# B&R Automation Studio project Kontrol (part 2)

#### Cyclic.st
```iecst
PROGRAM _CYCLIC

	//-------------------------------------------------------------------------------------------
	(*Parametros*)
	IF link_mdb_parametros.NewValue THEN
		link_mdb_parametros.NewValue    := FALSE;
	//-------------------------------------------------------------------------------------------

		UG.Parametro.UP_Partindo_Tempo := MDB_Parametros[1];
		UG.Parametro.UPGM_Partindo_Tempo := MDB_Parametros[2];
		UG.Parametro.UMVD_Partindo_Tempo := MDB_Parametros[3];
		UG.Parametro.UPS_Partindo_Tempo := MDB_Parametros[4];
		UG.Parametro.US_Parando_Tempo := MDB_Parametros[5];
		UG.Parametro.UPS_Parando_Tempo := MDB_Parametros[6];
		UG.Parametro.UMVD_Parando_Tempo := MDB_Parametros[7];
		UG.Parametro.UPGM_Parando_Tempo := MDB_Parametros[8];
		UG.Parametro.UPGM_Fechar_FA_Tempo := MDB_Parametros[9];
		//0.0 := MDB_Parametros[10];
		//0.0 := MDB_Parametros[11];
		//0.0 := MDB_Parametros[12];
		//0.0 := MDB_Parametros[13];
		//0.0 := MDB_Parametros[14];
		//0.0 := MDB_Parametros[15];
		//0.0 := MDB_Parametros[16];
		//0.0 := MDB_Parametros[17];
		//0.0 := MDB_Parametros[18];
		//0.0 := MDB_Parametros[19];
		//0.0 := MDB_Parametros[20];
		SFA.Parametro.Delta_Pressao.SensorMin := MDB_Parametros[21];
		SFA.Parametro.Delta_Pressao.SensorMax := MDB_Parametros[22];
		SFA.Parametro.Delta_Pressao.Alarme := MDB_Parametros[23];
		SFA.Parametro.Delta_Pressao.Trip := MDB_Parametros[24];
		SFA.Parametro.Delta_Pressao.Tempo_AL := MDB_Parametros[25];
		SFA.Parametro.Delta_Pressao.Tempo_TR := MDB_Parametros[26];
		SFA.Parametro.Pressao1_Lado_Limpo.SensorMin := MDB_Parametros[27];
		SFA.Parametro.Pressao1_Lado_Limpo.SensorMax := MDB_Parametros[28];
		SFA.Parametro.Pressao1_Lado_Limpo.Alarme := MDB_Parametros[29];
		SFA.Parametro.Pressao1_Lado_Limpo.Trip := MDB_Parametros[30];
		SFA.Parametro.Pressao1_Lado_Limpo.Tempo_AL := MDB_Parametros[31];
		SFA.Parametro.Pressao1_Lado_Limpo.Tempo_TR := MDB_Parametros[32];
		SFA.Parametro.Pressao2_Lado_Limpo.SensorMin := MDB_Parametros[33];
		SFA.Parametro.Pressao2_Lado_Limpo.SensorMax := MDB_Parametros[34];
		SFA.Parametro.Pressao2_Lado_Limpo.Alarme := MDB_Parametros[35];
		SFA.Parametro.Pressao2_Lado_Limpo.Trip := MDB_Parametros[36];
		SFA.Parametro.Pressao2_Lado_Limpo.Tempo_AL := MDB_Parametros[37];
		SFA.Parametro.Pressao2_Lado_Limpo.Tempo_TR := MDB_Parametros[38];
		SFA.Parametro.Pressao1_Lado_Sujo.SensorMin := MDB_Parametros[39];
		SFA.Parametro.Pressao1_Lado_Sujo.SensorMax := MDB_Parametros[40];
		SFA.Parametro.Pressao1_Lado_Sujo.Alarme := MDB_Parametros[41];
		SFA.Parametro.Pressao1_Lado_Sujo.Trip := MDB_Parametros[42];
		SFA.Parametro.Pressao1_Lado_Sujo.Tempo_AL := MDB_Parametros[43];
		SFA.Parametro.Pressao1_Lado_Sujo.Tempo_TR := MDB_Parametros[44];
		SFA.Parametro.Pressao2_Lado_Sujo.SensorMin := MDB_Parametros[45];
		SFA.Parametro.Pressao2_Lado_Sujo.SensorMax := MDB_Parametros[46];
		SFA.Parametro.Pressao2_Lado_Sujo.Alarme := MDB_Parametros[47];
		SFA.Parametro.Pressao2_Lado_Sujo.Trip := MDB_Parametros[48];
		SFA.Parametro.Pressao2_Lado_Sujo.Tempo_AL := MDB_Parametros[49];
		SFA.Parametro.Pressao2_Lado_Sujo.Tempo_TR := MDB_Parametros[50];
		SFA.Parametro.Filtro1_Tempo_Trabalho := MDB_Parametros[51];
		SFA.Parametro.Filtro1_Tempo_Lavagem := MDB_Parametros[52];
		SFA.Parametro.Filtro1_Tempo_Abrir_Filtro_Limpo := MDB_Parametros[53];
		SFA.Parametro.Filtro1_Tempo_Fechar_Filtro_Sujo := MDB_Parametros[54];
		SFA.Parametro.Filtro2_Tempo_Trabalho := MDB_Parametros[55];
		SFA.Parametro.Filtro2_Tempo_Lavagem := MDB_Parametros[56];
		SFA.Parametro.Filtro2_Tempo_Abrir_Filtro_Limpo := MDB_Parametros[57];
		SFA.Parametro.Filtro2_Tempo_Fechar_Filtro_Sujo := MDB_Parametros[58];
		SFA.Parametro.Filtro1_Delta_Retrolav := MDB_Parametros[59]; //delta de pressão para retrolavagem filtro 1
		SFA.Parametro.Filtro2_Delta_Retrolav := MDB_Parametros[60]; //delta de pressão para retrolavagem filtro 2
		//0.0 := MDB_Parametros[61];
		//0.0 := MDB_Parametros[62];
		//0.0 := MDB_Parametros[63];
		//0.0 := MDB_Parametros[64];
		//0.0 := MDB_Parametros[65];
		//0.0 := MDB_Parametros[66];
		//0.0 := MDB_Parametros[67];
		//0.0 := MDB_Parametros[68];
		//0.0 := MDB_Parametros[69];
		//0.0 := MDB_Parametros[70];
		UHLM.Parametro.Temperatura.SensorMin := MDB_Parametros[71];
		UHLM.Parametro.Temperatura.SensorMax := MDB_Parametros[72];
		UHLM.Parametro.Temperatura.Alarme := MDB_Parametros[73];
		UHLM.Parametro.Temperatura.Trip := MDB_Parametros[74];
		UHLM.Parametro.Temperatura.Tempo_AL := MDB_Parametros[75];
		UHLM.Parametro.Temperatura.Tempo_TR := MDB_Parametros[76];
		UHLM.Parametro.Vazao.SensorMin := MDB_Parametros[77];
		UHLM.Parametro.Vazao.SensorMax := MDB_Parametros[78];
		UHLM.Parametro.Vazao.Alarme := MDB_Parametros[79];
		UHLM.Parametro.Vazao.Trip := MDB_Parametros[80];
		UHLM.Parametro.Vazao.Tempo_AL := MDB_Parametros[81];
		UHLM.Parametro.Vazao.Tempo_TR := MDB_Parametros[82];
		UHLM.Parametro.Ventilador.Ligar := MDB_Parametros[83];
		UHLM.Parametro.Ventilador.Desligar := MDB_Parametros[84];
		//0.0 := MDB_Parametros[85];
		//0.0 := MDB_Parametros[86];
		//0.0 := MDB_Parametros[87];
		//0.0 := MDB_Parametros[88];
		//0.0 := MDB_Parametros[89];
		//0.0 := MDB_Parametros[90];
		//0.0 := MDB_Parametros[91];
		//0.0 := MDB_Parametros[92];
		//0.0 := MDB_Parametros[93];
		//0.0 := MDB_Parametros[94];
		//0.0 := MDB_Parametros[95];
		//0.0 := MDB_Parametros[96];
		//0.0 := MDB_Parametros[97];
		//0.0 := MDB_Parametros[98];
		//0.0 := MDB_Parametros[99];
		//0.0 := MDB_Parametros[100];
		UHRV.Parametro.Temperatura.SensorMin := MDB_Parametros[101];
		UHRV.Parametro.Temperatura.SensorMax := MDB_Parametros[102];
		UHRV.Parametro.Temperatura.Alarme := MDB_Parametros[103];
		UHRV.Parametro.Temperatura.Trip := MDB_Parametros[104];
		UHRV.Parametro.Temperatura.Tempo_AL := MDB_Parametros[105];
		UHRV.Parametro.Temperatura.Tempo_TR := MDB_Parametros[106];
		UHRV.Parametro.Pressao.SensorMin := MDB_Parametros[107];
		UHRV.Parametro.Pressao.SensorMax := MDB_Parametros[108];
		UHRV.Parametro.Pressao.Alarme := MDB_Parametros[109];
		UHRV.Parametro.Pressao.Trip := MDB_Parametros[110];
		UHRV.Parametro.Pressao.Tempo_AL := MDB_Parametros[111];
		UHRV.Parametro.Pressao.Tempo_TR := MDB_Parametros[112];
		UHRV.Parametro.Pressao.Normal_Min := MDB_Parametros[113];
		UHRV.Parametro.Pressao.Normal_Max := MDB_Parametros[114];
		UHRV.Parametro.Tempo_Pressurizar := MDB_Parametros[115];
		//0.0 := MDB_Parametros[116];
		//0.0 := MDB_Parametros[117];
		//0.0 := MDB_Parametros[118];
		//0.0 := MDB_Parametros[119];
		//0.0 := MDB_Parametros[120];
		//0.0 := MDB_Parametros[121];
		//0.0 := MDB_Parametros[122];
		//0.0 := MDB_Parametros[123];
		//0.0 := MDB_Parametros[124];
		//0.0 := MDB_Parametros[125];
		//0.0 := MDB_Parametros[126];
		//0.0 := MDB_Parametros[127];
		//0.0 := MDB_Parametros[128];
		//0.0 := MDB_Parametros[129];
		//0.0 := MDB_Parametros[130];
		Freio.Parametro.Tempo_Aplicado := MDB_Parametros[131];
		Freio.Parametro.Tempo_Desaplicado := MDB_Parametros[132];
		//0.0 := MDB_Parametros[133];
		//0.0 := MDB_Parametros[134];
		//0.0 := MDB_Parametros[135];
		//0.0 := MDB_Parametros[136];
		//0.0 := MDB_Parametros[137];
		//0.0 := MDB_Parametros[138];
		//0.0 := MDB_Parametros[139];
		//0.0 := MDB_Parametros[140];
//		VByPass.Parametro.Tempo.Abrir := MDB_Parametros[141];
//		VByPass.Parametro.Tempo.Fechar := MDB_Parametros[142];
		//0.0 := MDB_Parametros[143];
		//0.0 := MDB_Parametros[144];
		//0.0 := MDB_Parametros[145];
		//0.0 := MDB_Parametros[146];
		//0.0 := MDB_Parametros[147];
		//0.0 := MDB_Parametros[148];
		//0.0 := MDB_Parametros[149];
		//0.0 := MDB_Parametros[150];
//		VBorb.Parametro.Tempo.Abrir := MDB_Parametros[151];
//		VBorb.Parametro.Tempo.Fechar := MDB_Parametros[152];
//		VBorb.Parametro.Tempo.Equalizar := MDB_Parametros[153];
//		VBorb.Parametro.Delta_Pressao := MDB_Parametros[154];
//		VBorb.Parametro.Pressao.Montante.SensorMin := MDB_Parametros[155];
//		VBorb.Parametro.Pressao.Montante.SensorMax := MDB_Parametros[156];
//		VBorb.Parametro.Pressao.Jusante.SensorMin := MDB_Parametros[157];
//		VBorb.Parametro.Pressao.Jusante.SensorMax := MDB_Parametros[158];
		//0.0 := MDB_Parametros[159];
		//0.0 := MDB_Parametros[160];
		//0.0 := MDB_Parametros[161];
		//0.0 := MDB_Parametros[162];
		//0.0 := MDB_Parametros[163];
		//0.0 := MDB_Parametros[164];
		//0.0 := MDB_Parametros[165];
		//0.0 := MDB_Parametros[166];
		//0.0 := MDB_Parametros[167];
		Comporta1.Parametro.Encoder1_SensorMin := MDB_Parametros[168];
		Comporta1.Parametro.Encoder1_SensorMax := MDB_Parametros[169];
		Comporta1.Parametro.Tempo_Cracking := MDB_Parametros[170];
		Comporta1.Parametro.Tempo_Falha_Abertura := MDB_Parametros[171];
		Comporta1.Parametro.Tempo_Falha_Cracking := MDB_Parametros[172];
		Comporta1.Parametro.Tempo_Falha_Fechando := MDB_Parametros[173];
		Comporta1.Parametro.Tempo_Falha_Reposicao := MDB_Parametros[174];
//		Comporta.Parametro.Pressao.Montante.SensorMin := MDB_Parametros[175];
//		Comporta.Parametro.Pressao.Montante.SensorMax := MDB_Parametros[176];
		Comporta2.Parametro.Encoder2_SensorMin := MDB_Parametros[177];
		Comporta2.Parametro.Encoder2_SensorMax := MDB_Parametros[178];
		Comporta2.Parametro.Tempo_Cracking := MDB_Parametros[179];
		Comporta2.Parametro.Tempo_Falha_Abertura := MDB_Parametros[180];
		Comporta2.Parametro.Tempo_Falha_Cracking := MDB_Parametros[181];
		Comporta2.Parametro.Tempo_Falha_Fechando := MDB_Parametros[182];
		Comporta2.Parametro.Tempo_Falha_Reposicao := MDB_Parametros[183];
		Comporta_UH.Parametro.Temperatura_Oleo.SensorMin := MDB_Parametros[184];
		Comporta_UH.Parametro.Temperatura_Oleo.SensorMax := MDB_Parametros[185];
		Comporta_UH.Parametro.Temperatura_Oleo.Alarme := MDB_Parametros[186];
		Comporta_UH.Parametro.Temperatura_Oleo.Trip := MDB_Parametros[187];
		Comporta_UH.Parametro.Temperatura_Oleo.Tempo_AL := MDB_Parametros[188];
		Comporta_UH.Parametro.Temperatura_Oleo.Tempo_TR := MDB_Parametros[189];
		//0.0 := MDB_Parametros[190];
		Turbina.Parametro.Gaxeteiro.Temperatura.SensorMin := MDB_Parametros[191];
		Turbina.Parametro.Gaxeteiro.Temperatura.SensorMax := MDB_Parametros[192];
		Turbina.Parametro.Gaxeteiro.Temperatura.Alarme := MDB_Parametros[193];
		Turbina.Parametro.Gaxeteiro.Temperatura.Trip := MDB_Parametros[194];
		Turbina.Parametro.Gaxeteiro.Temperatura.Tempo_AL := MDB_Parametros[195];
		Turbina.Parametro.Gaxeteiro.Temperatura.Tempo_TR := MDB_Parametros[196];
		Turbina.Parametro.Mancal1.Temperatura.SensorMin := MDB_Parametros[197];
		Turbina.Parametro.Mancal1.Temperatura.SensorMax := MDB_Parametros[198];
		Turbina.Parametro.Mancal1.Temperatura.Alarme := MDB_Parametros[199];
		Turbina.Parametro.Mancal1.Temperatura.Trip := MDB_Parametros[200];
		Turbina.Parametro.Mancal1.Temperatura.Tempo_AL := MDB_Parametros[201];
		Turbina.Parametro.Mancal1.Temperatura.Tempo_TR := MDB_Parametros[202];
		Turbina.Parametro.Mancal2.Temperatura.SensorMin := MDB_Parametros[203];
		Turbina.Parametro.Mancal2.Temperatura.SensorMax := MDB_Parametros[204];
		Turbina.Parametro.Mancal2.Temperatura.Alarme := MDB_Parametros[205];
		Turbina.Parametro.Mancal2.Temperatura.Trip := MDB_Parametros[206];
		Turbina.Parametro.Mancal2.Temperatura.Tempo_AL := MDB_Parametros[207];
		Turbina.Parametro.Mancal2.Temperatura.Tempo_TR := MDB_Parametros[208];
		Turbina.Parametro.Mancal3.Temperatura.SensorMin := MDB_Parametros[209];
		Turbina.Parametro.Mancal3.Temperatura.SensorMax := MDB_Parametros[210];
		Turbina.Parametro.Mancal3.Temperatura.Alarme := MDB_Parametros[211];
		Turbina.Parametro.Mancal3.Temperatura.Trip := MDB_Parametros[212];
		Turbina.Parametro.Mancal3.Temperatura.Tempo_AL := MDB_Parametros[213];
		Turbina.Parametro.Mancal3.Temperatura.Tempo_TR := MDB_Parametros[214];
		Turbina.Parametro.Mancal4.Temperatura.SensorMin := MDB_Parametros[215];
		Turbina.Parametro.Mancal4.Temperatura.SensorMax := MDB_Parametros[216];
		Turbina.Parametro.Mancal4.Temperatura.Alarme := MDB_Parametros[217];
		Turbina.Parametro.Mancal4.Temperatura.Trip := MDB_Parametros[218];
		Turbina.Parametro.Mancal4.Temperatura.Tempo_AL := MDB_Parametros[219];
		Turbina.Parametro.Mancal4.Temperatura.Tempo_TR := MDB_Parametros[220];
		Turbina.Parametro.Mancal5.Temperatura.SensorMin := MDB_Parametros[221];
		Turbina.Parametro.Mancal5.Temperatura.SensorMax := MDB_Parametros[222];
		Turbina.Parametro.Mancal5.Temperatura.Alarme := MDB_Parametros[223];
		Turbina.Parametro.Mancal5.Temperatura.Trip := MDB_Parametros[224];
		Turbina.Parametro.Mancal5.Temperatura.Tempo_AL := MDB_Parametros[225];
		Turbina.Parametro.Mancal5.Temperatura.Tempo_TR := MDB_Parametros[226];
		Turbina.Parametro.Mancal6.Temperatura.SensorMin := MDB_Parametros[227];
		Turbina.Parametro.Mancal6.Temperatura.SensorMax := MDB_Parametros[228];
		Turbina.Parametro.Mancal6.Temperatura.Alarme := MDB_Parametros[229];
		Turbina.Parametro.Mancal6.Temperatura.Trip := MDB_Parametros[230];
		Turbina.Parametro.Mancal6.Temperatura.Tempo_AL := MDB_Parametros[231];
		Turbina.Parametro.Mancal6.Temperatura.Tempo_TR := MDB_Parametros[232];
		Turbina.Parametro.CaixaEspiral.Pressao.SensorMin := MDB_Parametros[233];
		Turbina.Parametro.CaixaEspiral.Pressao.SensorMax := MDB_Parametros[234];
		Turbina.Parametro.CaixaEspiral.Pressao.Alarme := MDB_Parametros[235];
		Turbina.Parametro.CaixaEspiral.Pressao.Trip := MDB_Parametros[236];
		Turbina.Parametro.CaixaEspiral.Pressao.Tempo_AL := MDB_Parametros[237];
		Turbina.Parametro.CaixaEspiral.Pressao.Tempo_TR := MDB_Parametros[238];
		Turbina.Parametro.Delta_Pressao := MDB_Parametros[239];
		//0.0 := MDB_Parametros[240];
		//0.0 := MDB_Parametros[241];
		//0.0 := MDB_Parametros[242];
		//0.0 := MDB_Parametros[243];
		//0.0 := MDB_Parametros[244];
		//0.0 := MDB_Parametros[245];
		//0.0 := MDB_Parametros[246];
		//0.0 := MDB_Parametros[247];
		//0.0 := MDB_Parametros[248];
		//0.0 := MDB_Parametros[249];
		//0.0 := MDB_Parametros[250];
		Gerador.Parametro.Fase_A.Temperatura.SensorMin := MDB_Parametros[251];
		Gerador.Parametro.Fase_A.Temperatura.SensorMax := MDB_Parametros[252];
		Gerador.Parametro.Fase_A.Temperatura.Alarme := MDB_Parametros[253];
		Gerador.Parametro.Fase_A.Temperatura.Trip := MDB_Parametros[254];
		Gerador.Parametro.Fase_A.Temperatura.Tempo_AL := MDB_Parametros[255];
		Gerador.Parametro.Fase_A.Temperatura.Tempo_TR := MDB_Parametros[256];
		Gerador.Parametro.Fase_B.Temperatura.SensorMin := MDB_Parametros[257];
		Gerador.Parametro.Fase_B.Temperatura.SensorMax := MDB_Parametros[258];
		Gerador.Parametro.Fase_B.Temperatura.Alarme := MDB_Parametros[259];
		Gerador.Parametro.Fase_B.Temperatura.Trip := MDB_Parametros[260];
		Gerador.Parametro.Fase_B.Temperatura.Tempo_AL := MDB_Parametros[261];
		Gerador.Parametro.Fase_B.Temperatura.Tempo_TR := MDB_Parametros[262];
		Gerador.Parametro.Fase_C.Temperatura.SensorMin := MDB_Parametros[263];
		Gerador.Parametro.Fase_C.Temperatura.SensorMax := MDB_Parametros[264];
		Gerador.Parametro.Fase_C.Temperatura.Alarme := MDB_Parametros[265];
		Gerador.Parametro.Fase_C.Temperatura.Trip := MDB_Parametros[266];
		Gerador.Parametro.Fase_C.Temperatura.Tempo_AL := MDB_Parametros[267];
		Gerador.Parametro.Fase_C.Temperatura.Tempo_TR := MDB_Parametros[268];
		Gerador.Parametro.NucleoEstatorico1.Temperatura.SensorMin := MDB_Parametros[269];
		Gerador.Parametro.NucleoEstatorico1.Temperatura.SensorMax := MDB_Parametros[270];
		Gerador.Parametro.NucleoEstatorico1.Temperatura.Alarme := MDB_Parametros[271];
		Gerador.Parametro.NucleoEstatorico1.Temperatura.Trip := MDB_Parametros[272];
		Gerador.Parametro.NucleoEstatorico1.Temperatura.Tempo_AL := MDB_Parametros[273];
		Gerador.Parametro.NucleoEstatorico1.Temperatura.Tempo_TR := MDB_Parametros[274];
		Gerador.Parametro.NucleoEstatorico2.Temperatura.SensorMin := MDB_Parametros[275];
		Gerador.Parametro.NucleoEstatorico2.Temperatura.SensorMax := MDB_Parametros[276];
		Gerador.Parametro.NucleoEstatorico2.Temperatura.Alarme := MDB_Parametros[277];
		Gerador.Parametro.NucleoEstatorico2.Temperatura.Trip := MDB_Parametros[278];
		Gerador.Parametro.NucleoEstatorico2.Temperatura.Tempo_AL := MDB_Parametros[279];
		Gerador.Parametro.NucleoEstatorico2.Temperatura.Tempo_TR := MDB_Parametros[280];
		Gerador.Parametro.NucleoEstatorico3.Temperatura.SensorMin := MDB_Parametros[281];
		Gerador.Parametro.NucleoEstatorico3.Temperatura.SensorMax := MDB_Parametros[282];
		Gerador.Parametro.NucleoEstatorico3.Temperatura.Alarme := MDB_Parametros[283];
		Gerador.Parametro.NucleoEstatorico3.Temperatura.Trip := MDB_Parametros[284];
		Gerador.Parametro.NucleoEstatorico3.Temperatura.Tempo_AL := MDB_Parametros[285];
		Gerador.Parametro.NucleoEstatorico3.Temperatura.Tempo_TR := MDB_Parametros[286];
		Gerador.Parametro.Mancal1.Temperatura.SensorMin := MDB_Parametros[287];
		Gerador.Parametro.Mancal1.Temperatura.SensorMax := MDB_Parametros[288];
		Gerador.Parametro.Mancal1.Temperatura.Alarme := MDB_Parametros[289];
		Gerador.Parametro.Mancal1.Temperatura.Trip := MDB_Parametros[290];
		Gerador.Parametro.Mancal1.Temperatura.Tempo_AL := MDB_Parametros[291];
		Gerador.Parametro.Mancal1.Temperatura.Tempo_TR := MDB_Parametros[292];
		Gerador.Parametro.Mancal2.Temperatura.SensorMin := MDB_Parametros[293];
		Gerador.Parametro.Mancal2.Temperatura.SensorMax := MDB_Parametros[294];
		Gerador.Parametro.Mancal2.Temperatura.Alarme := MDB_Parametros[295];
		Gerador.Parametro.Mancal2.Temperatura.Trip := MDB_Parametros[296];
		Gerador.Parametro.Mancal2.Temperatura.Tempo_AL := MDB_Parametros[297];
		Gerador.Parametro.Mancal2.Temperatura.Tempo_TR := MDB_Parametros[298];
		Gerador.Parametro.Mancal3.Temperatura.SensorMin := MDB_Parametros[299];
		Gerador.Parametro.Mancal3.Temperatura.SensorMax := MDB_Parametros[300];
		Gerador.Parametro.Mancal3.Temperatura.Alarme := MDB_Parametros[301];
		Gerador.Parametro.Mancal3.Temperatura.Trip := MDB_Parametros[302];
		Gerador.Parametro.Mancal3.Temperatura.Tempo_AL := MDB_Parametros[303];
		Gerador.Parametro.Mancal3.Temperatura.Tempo_TR := MDB_Parametros[304];
		Gerador.Parametro.Mancal4.Temperatura.SensorMin := MDB_Parametros[305];
		Gerador.Parametro.Mancal4.Temperatura.SensorMax := MDB_Parametros[306];
		Gerador.Parametro.Mancal4.Temperatura.Alarme := MDB_Parametros[307];
		Gerador.Parametro.Mancal4.Temperatura.Trip := MDB_Parametros[308];
		Gerador.Parametro.Mancal4.Temperatura.Tempo_AL := MDB_Parametros[309];
		Gerador.Parametro.Mancal4.Temperatura.Tempo_TR := MDB_Parametros[310];
		Gerador.Parametro.Mancal5.Temperatura.SensorMin := MDB_Parametros[311];
		Gerador.Parametro.Mancal5.Temperatura.SensorMax := MDB_Parametros[312];
		Gerador.Parametro.Mancal5.Temperatura.Alarme := MDB_Parametros[313];
		Gerador.Parametro.Mancal5.Temperatura.Trip := MDB_Parametros[314];
		Gerador.Parametro.Mancal5.Temperatura.Tempo_AL := MDB_Parametros[315];
		Gerador.Parametro.Mancal5.Temperatura.Tempo_TR := MDB_Parametros[316];
		Gerador.Parametro.Mancal6.Temperatura.SensorMin := MDB_Parametros[317];
		Gerador.Parametro.Mancal6.Temperatura.SensorMax := MDB_Parametros[318];
		Gerador.Parametro.Mancal6.Temperatura.Alarme := MDB_Parametros[319];
		Gerador.Parametro.Mancal6.Temperatura.Trip := MDB_Parametros[320];
		Gerador.Parametro.Mancal6.Temperatura.Tempo_AL := MDB_Parametros[321];
		Gerador.Parametro.Mancal6.Temperatura.Tempo_TR := MDB_Parametros[322];
		//0.0 := MDB_Parametros[323];
		//0.0 := MDB_Parametros[324];
		//0.0 := MDB_Parametros[325];
		//0.0 := MDB_Parametros[326];
		//0.0 := MDB_Parametros[327];
		//0.0 := MDB_Parametros[328];
		//0.0 := MDB_Parametros[329];
		//0.0 := MDB_Parametros[330];
		//0.0 := MDB_Parametros[331];
		//0.0 := MDB_Parametros[332];
		//0.0 := MDB_Parametros[333];
		//0.0 := MDB_Parametros[334];
		//0.0 := MDB_Parametros[335];
		//0.0 := MDB_Parametros[336];
		//0.0 := MDB_Parametros[337];
		//0.0 := MDB_Parametros[338];
		//0.0 := MDB_Parametros[339];
		//0.0 := MDB_Parametros[340];
		RT.Parametro.PWR.Temperatura.SensorMin := MDB_Parametros[341];
		RT.Parametro.PWR.Temperatura.SensorMax := MDB_Parametros[342];
		RT.Parametro.PWR.Temperatura.Alarme := MDB_Parametros[343];
		RT.Parametro.PWR.Temperatura.Trip := MDB_Parametros[344];
		RT.Parametro.PWR.Temperatura.Tempo_AL := MDB_Parametros[345];
		RT.Parametro.PWR.Temperatura.Tempo_TR := MDB_Parametros[346];
		//0.0 := MDB_Parametros[347];
		//0.0 := MDB_Parametros[348];
		//0.0 := MDB_Parametros[349];
		//0.0 := MDB_Parametros[350];
		//0.0 := MDB_Parametros[351];
		//0.0 := MDB_Parametros[352];
		//0.0 := MDB_Parametros[353];
		//0.0 := MDB_Parametros[354];
		//0.0 := MDB_Parametros[355];
		//0.0 := MDB_Parametros[356];
		//0.0 := MDB_Parametros[357];
		//0.0 := MDB_Parametros[358];
		//0.0 := MDB_Parametros[359];
		//0.0 := MDB_Parametros[360];
		Trafo_Exc.Parametro.Fase_A.Temperatura.SensorMin := MDB_Parametros[361];
		Trafo_Exc.Parametro.Fase_A.Temperatura.SensorMax := MDB_Parametros[362];
		Trafo_Exc.Parametro.Fase_A.Temperatura.Alarme := MDB_Parametros[363];
		Trafo_Exc.Parametro.Fase_A.Temperatura.Trip := MDB_Parametros[364];
		Trafo_Exc.Parametro.Fase_A.Temperatura.Tempo_AL := MDB_Parametros[365];
		Trafo_Exc.Parametro.Fase_A.Temperatura.Tempo_TR := MDB_Parametros[366];
		Trafo_Exc.Parametro.Fase_B.Temperatura.SensorMin := MDB_Parametros[367];
		Trafo_Exc.Parametro.Fase_B.Temperatura.SensorMax := MDB_Parametros[368];
		Trafo_Exc.Parametro.Fase_B.Temperatura.Alarme := MDB_Parametros[369];
		Trafo_Exc.Parametro.Fase_B.Temperatura.Trip := MDB_Parametros[370];
		Trafo_Exc.Parametro.Fase_B.Temperatura.Tempo_AL := MDB_Parametros[371];
		Trafo_Exc.Parametro.Fase_B.Temperatura.Tempo_TR := MDB_Parametros[372];
		Trafo_Exc.Parametro.Fase_C.Temperatura.SensorMin := MDB_Parametros[373];
		Trafo_Exc.Parametro.Fase_C.Temperatura.SensorMax := MDB_Parametros[374];
		Trafo_Exc.Parametro.Fase_C.Temperatura.Alarme := MDB_Parametros[375];
		Trafo_Exc.Parametro.Fase_C.Temperatura.Trip := MDB_Parametros[376];
		Trafo_Exc.Parametro.Fase_C.Temperatura.Tempo_AL := MDB_Parametros[377];
		Trafo_Exc.Parametro.Fase_C.Temperatura.Tempo_TR := MDB_Parametros[378];
		//0.0 := MDB_Parametros[379];
		//0.0 := MDB_Parametros[380];
		//0.0 := MDB_Parametros[381];
		//0.0 := MDB_Parametros[382];
		//0.0 := MDB_Parametros[383];
		//0.0 := MDB_Parametros[384];
		//0.0 := MDB_Parametros[385];
		//0.0 := MDB_Parametros[386];
		//0.0 := MDB_Parametros[387];
		//0.0 := MDB_Parametros[388];
		//0.0 := MDB_Parametros[389];
		//0.0 := MDB_Parametros[390];
		Nivel.Parametro.Nivel_Ligar := MDB_Parametros[391];
		Nivel.Parametro.Nivel_Desligar := MDB_Parametros[392];
		Nivel.Parametro.Nivel_Trip := MDB_Parametros[393];
		Nivel.Parametro.Nivel_Min := MDB_Parametros[394];
		Nivel.Parametro.Nivel_Max := MDB_Parametros[395];
		Nivel.Parametro.Potencia_Min := MDB_Parametros[396];
		Nivel.Parametro.Potencia_Max := MDB_Parametros[397];
		Nivel.Parametro.PID.Kp := MDB_Parametros[398];
		Nivel.Parametro.PID.Ki := MDB_Parametros[399];
		Nivel.Parametro.PID.Kd := MDB_Parametros[400];
		Nivel.Parametro.PID.Tf := MDB_Parametros[401];
		//0.0 := MDB_Parametros[402];
		//0.0 := MDB_Parametros[403];
		//0.0 := MDB_Parametros[404];
		//0.0 := MDB_Parametros[405];
		//0.0 := MDB_Parametros[406];
		//0.0 := MDB_Parametros[407];
		//0.0 := MDB_Parametros[408];
		//0.0 := MDB_Parametros[409];
		//0.0 := MDB_Parametros[410];
		Nivel.Parametro.Barragem.SensorMin := MDB_Parametros[411];
		Nivel.Parametro.Barragem.SensorMax := MDB_Parametros[412];
		//0.0 := MDB_Parametros[413];
		//0.0 := MDB_Parametros[414];
		Nivel.Parametro.Barragem.Alarme := MDB_Parametros[415];
		Nivel.Parametro.Barragem.Trip := MDB_Parametros[416];
		Nivel.Parametro.Barragem.Tempo_AL := MDB_Parametros[417];
		Nivel.Parametro.Barragem.Tempo_TR := MDB_Parametros[418];
		Nivel.Parametro.Jusante.SensorMin := MDB_Parametros[419];
		Nivel.Parametro.Jusante.SensorMax := MDB_Parametros[420];
		//0.0 := MDB_Parametros[421];
		Nivel.Parametro.Jusante.Cota := MDB_Parametros[422];
		Nivel.Parametro.Jusante.Alarme := MDB_Parametros[423];
		Nivel.Parametro.Jusante.Trip := MDB_Parametros[424];
		Nivel.Parametro.Jusante.Tempo_AL := MDB_Parametros[425];
		Nivel.Parametro.Jusante.Tempo_TR := MDB_Parametros[426];
		//0.0 := MDB_Parametros[427];
		//0.0 := MDB_Parametros[428];
		//0.0 := MDB_Parametros[429];
		Nivel.Parametro.Jusante_Grade1.SensorMin := MDB_Parametros[430];
		Nivel.Parametro.Jusante_Grade1.SensorMax := MDB_Parametros[431];
		Nivel.Parametro.Jusante_Grade1.Cota := MDB_Parametros[432];
		Nivel.Parametro.Jusante_Grade1.Alarme := MDB_Parametros[433];
		Nivel.Parametro.Jusante_Grade1.Trip := MDB_Parametros[434];
		Nivel.Parametro.Jusante_Grade1.Tempo_AL := MDB_Parametros[435];
		Nivel.Parametro.Jusante_Grade1.Tempo_TR := MDB_Parametros[436];
		//0.0 := MDB_Parametros[437];
		//0.0 := MDB_Parametros[438];
		//0.0 := MDB_Parametros[439];
		Nivel.Parametro.Jusante_Grade2.SensorMin := MDB_Parametros[440];
		Nivel.Parametro.Jusante_Grade2.SensorMax := MDB_Parametros[441];
		Nivel.Parametro.Jusante_Grade2.Cota := MDB_Parametros[442];
		Nivel.Parametro.Jusante_Grade2.Alarme := MDB_Parametros[443];
		Nivel.Parametro.Jusante_Grade2.Trip := MDB_Parametros[444];
		Nivel.Parametro.Jusante_Grade2.Tempo_AL := MDB_Parametros[445];
		Nivel.Parametro.Jusante_Grade2.Tempo_TR := MDB_Parametros[446];
		//0.0 := MDB_Parametros[447];
		//0.0 := MDB_Parametros[448];
		//0.0 := MDB_Parametros[449];
		//0.0 := MDB_Parametros[450];
		//0.0 := MDB_Parametros[451];
		//0.0 := MDB_Parametros[452];
		//0.0 := MDB_Parametros[453];
		//0.0 := MDB_Parametros[454];
		//0.0 := MDB_Parametros[455];
		//0.0 := MDB_Parametros[456];
		//0.0 := MDB_Parametros[457];
		//0.0 := MDB_Parametros[458];
		//0.0 := MDB_Parametros[459];
		//0.0 := MDB_Parametros[460];

	//-------------------------------------------------------------------------------------------

	ELSE

	//-------------------------------------------------------------------------------------------

		MDB_Parametros[1]:=UG.Parametro.UP_Partindo_Tempo;
		MDB_Parametros[2]:=UG.Parametro.UPGM_Partindo_Tempo;
		MDB_Parametros[3]:=UG.Parametro.UMVD_Partindo_Tempo;
		MDB_Parametros[4]:=UG.Parametro.UPS_Partindo_Tempo;
		MDB_Parametros[5]:=UG.Parametro.US_Parando_Tempo;
		MDB_Parametros[6]:=UG.Parametro.UPS_Parando_Tempo;
		MDB_Parametros[7]:=UG.Parametro.UMVD_Parando_Tempo;
		MDB_Parametros[8]:=UG.Parametro.UPGM_Parando_Tempo;
		MDB_Parametros[9]:=UG.Parametro.UPGM_Fechar_FA_Tempo;
		MDB_Parametros[10]:=0.0;
		MDB_Parametros[11]:=0.0;
		MDB_Parametros[12]:=0.0;
		MDB_Parametros[13]:=0.0;
		MDB_Parametros[14]:=0.0;
		MDB_Parametros[15]:=0.0;
		MDB_Parametros[16]:=0.0;
		MDB_Parametros[17]:=0.0;
		MDB_Parametros[18]:=0.0;
		MDB_Parametros[19]:=0.0;
		MDB_Parametros[20]:=0.0;
		MDB_Parametros[21]:=SFA.Parametro.Delta_Pressao.SensorMin;
		MDB_Parametros[22]:=SFA.Parametro.Delta_Pressao.SensorMax;
		MDB_Parametros[23]:=SFA.Parametro.Delta_Pressao.Alarme;
		MDB_Parametros[24]:=SFA.Parametro.Delta_Pressao.Trip;
		MDB_Parametros[25]:=SFA.Parametro.Delta_Pressao.Tempo_AL;
		MDB_Parametros[26]:=SFA.Parametro.Delta_Pressao.Tempo_TR;
		MDB_Parametros[27]:=SFA.Parametro.Pressao1_Lado_Limpo.SensorMin;
		MDB_Parametros[28]:=SFA.Parametro.Pressao1_Lado_Limpo.SensorMax;
		MDB_Parametros[29]:=SFA.Parametro.Pressao1_Lado_Limpo.Alarme;
		MDB_Parametros[30]:=SFA.Parametro.Pressao1_Lado_Limpo.Trip;
		MDB_Parametros[31]:=SFA.Parametro.Pressao1_Lado_Limpo.Tempo_AL;
		MDB_Parametros[32]:=SFA.Parametro.Pressao1_Lado_Limpo.Tempo_TR;
		MDB_Parametros[33]:=SFA.Parametro.Pressao2_Lado_Limpo.SensorMin;
		MDB_Parametros[34]:=SFA.Parametro.Pressao2_Lado_Limpo.SensorMax;
		MDB_Parametros[35]:=SFA.Parametro.Pressao2_Lado_Limpo.Alarme;
		MDB_Parametros[36]:=SFA.Parametro.Pressao2_Lado_Limpo.Trip;
		MDB_Parametros[37]:=SFA.Parametro.Pressao2_Lado_Limpo.Tempo_AL;
		MDB_Parametros[38]:=SFA.Parametro.Pressao2_Lado_Limpo.Tempo_TR;
		MDB_Parametros[39]:=SFA.Parametro.Pressao1_Lado_Sujo.SensorMin;
		MDB_Parametros[40]:=SFA.Parametro.Pressao1_Lado_Sujo.SensorMax;
		MDB_Parametros[41]:=SFA.Parametro.Pressao1_Lado_Sujo.Alarme;
		MDB_Parametros[42]:=SFA.Parametro.Pressao1_Lado_Sujo.Trip;
		MDB_Parametros[43]:=SFA.Parametro.Pressao1_Lado_Sujo.Tempo_AL;
		MDB_Parametros[44]:=SFA.Parametro.Pressao1_Lado_Sujo.Tempo_TR;
		MDB_Parametros[45]:=SFA.Parametro.Pressao2_Lado_Sujo.SensorMin;
		MDB_Parametros[46]:=SFA.Parametro.Pressao2_Lado_Sujo.SensorMax;
		MDB_Parametros[47]:=SFA.Parametro.Pressao2_Lado_Sujo.Alarme;
		MDB_Parametros[48]:=SFA.Parametro.Pressao2_Lado_Sujo.Trip;
		MDB_Parametros[49]:=SFA.Parametro.Pressao2_Lado_Sujo.Tempo_AL;
		MDB_Parametros[50]:=SFA.Parametro.Pressao2_Lado_Sujo.Tempo_TR;
		MDB_Parametros[51]:=SFA.Parametro.Filtro1_Tempo_Trabalho;
		MDB_Parametros[52]:=SFA.Parametro.Filtro1_Tempo_Lavagem;
		MDB_Parametros[53]:=SFA.Parametro.Filtro1_Tempo_Abrir_Filtro_Limpo;
		MDB_Parametros[54]:=SFA.Parametro.Filtro1_Tempo_Fechar_Filtro_Sujo;
		MDB_Parametros[55]:=SFA.Parametro.Filtro2_Tempo_Trabalho;
		MDB_Parametros[56]:=SFA.Parametro.Filtro2_Tempo_Lavagem;
		MDB_Parametros[57]:=SFA.Parametro.Filtro2_Tempo_Abrir_Filtro_Limpo;
		MDB_Parametros[58]:=SFA.Parametro.Filtro2_Tempo_Fechar_Filtro_Sujo;
		MDB_Parametros[59]:=SFA.Parametro.Filtro1_Delta_Retrolav;
		MDB_Parametros[60]:=SFA.Parametro.Filtro2_Delta_Retrolav;
		MDB_Parametros[61]:=0.0;
		MDB_Parametros[62]:=0.0;
		MDB_Parametros[63]:=0.0;
		MDB_Parametros[64]:=0.0;
		MDB_Parametros[65]:=0.0;
		MDB_Parametros[66]:=0.0;
		MDB_Parametros[67]:=0.0;
		MDB_Parametros[68]:=0.0;
		MDB_Parametros[69]:=0.0;
		MDB_Parametros[70]:=0.0;
		MDB_Parametros[71]:=UHLM.Parametro.Temperatura.SensorMin;
		MDB_Parametros[72]:=UHLM.Parametro.Temperatura.SensorMax;
		MDB_Parametros[73]:=UHLM.Parametro.Temperatura.Alarme;
		MDB_Parametros[74]:=UHLM.Parametro.Temperatura.Trip;
		MDB_Parametros[75]:=UHLM.Parametro.Temperatura.Tempo_AL;
		MDB_Parametros[76]:=UHLM.Parametro.Temperatura.Tempo_TR;
		MDB_Parametros[77]:=UHLM.Parametro.Vazao.SensorMin;
		MDB_Parametros[78]:=UHLM.Parametro.Vazao.SensorMax;
		MDB_Parametros[79]:=UHLM.Parametro.Vazao.Alarme;
		MDB_Parametros[80]:=UHLM.Parametro.Vazao.Trip;
		MDB_Parametros[81]:=UHLM.Parametro.Vazao.Tempo_AL;
		MDB_Parametros[82]:=UHLM.Parametro.Vazao.Tempo_TR;
		MDB_Parametros[83]:=UHLM.Parametro.Ventilador.Ligar;
		MDB_Parametros[84]:=UHLM.Parametro.Ventilador.Desligar;
		MDB_Parametros[85]:=0.0;
		MDB_Parametros[86]:=0.0;
		MDB_Parametros[87]:=0.0;
		MDB_Parametros[88]:=0.0;
		MDB_Parametros[89]:=0.0;
		MDB_Parametros[90]:=0.0;
		MDB_Parametros[91]:=0.0;
		MDB_Parametros[92]:=0.0;
		MDB_Parametros[93]:=0.0;
		MDB_Parametros[94]:=0.0;
		MDB_Parametros[95]:=0.0;
		MDB_Parametros[96]:=0.0;
		MDB_Parametros[97]:=0.0;
		MDB_Parametros[98]:=0.0;
		MDB_Parametros[99]:=0.0;
		MDB_Parametros[100]:=0.0;
		MDB_Parametros[101]:=UHRV.Parametro.Temperatura.SensorMin;
		MDB_Parametros[102]:=UHRV.Parametro.Temperatura.SensorMax;
		MDB_Parametros[103]:=UHRV.Parametro.Temperatura.Alarme;
		MDB_Parametros[104]:=UHRV.Parametro.Temperatura.Trip;
		MDB_Parametros[105]:=UHRV.Parametro.Temperatura.Tempo_AL;
		MDB_Parametros[106]:=UHRV.Parametro.Temperatura.Tempo_TR;
		MDB_Parametros[107]:=UHRV.Parametro.Pressao.SensorMin;
		MDB_Parametros[108]:=UHRV.Parametro.Pressao.SensorMax;
		MDB_Parametros[109]:=UHRV.Parametro.Pressao.Alarme;
		MDB_Parametros[110]:=UHRV.Parametro.Pressao.Trip;
		MDB_Parametros[111]:=UHRV.Parametro.Pressao.Tempo_AL;
		MDB_Parametros[112]:=UHRV.Parametro.Pressao.Tempo_TR;
		MDB_Parametros[113]:=UHRV.Parametro.Pressao.Normal_Min;
		MDB_Parametros[114]:=UHRV.Parametro.Pressao.Normal_Max;
		MDB_Parametros[115]:=UHRV.Parametro.Tempo_Pressurizar;
		MDB_Parametros[116]:=0.0;
		MDB_Parametros[117]:=0.0;
		MDB_Parametros[118]:=0.0;
		MDB_Parametros[119]:=0.0;
		MDB_Parametros[120]:=0.0;
		MDB_Parametros[121]:=0.0;
		MDB_Parametros[122]:=0.0;
		MDB_Parametros[123]:=0.0;
		MDB_Parametros[124]:=0.0;
		MDB_Parametros[125]:=0.0;
		MDB_Parametros[126]:=0.0;
		MDB_Parametros[127]:=0.0;
		MDB_Parametros[128]:=0.0;
		MDB_Parametros[129]:=0.0;
		MDB_Parametros[130]:=0.0;
		MDB_Parametros[131]:=Freio.Parametro.Tempo_Aplicado;
		MDB_Parametros[132]:=Freio.Parametro.Tempo_Desaplicado;
		MDB_Parametros[133]:=0.0;
		MDB_Parametros[134]:=0.0;
		MDB_Parametros[135]:=0.0;
		MDB_Parametros[136]:=0.0;
		MDB_Parametros[137]:=0.0;
		MDB_Parametros[138]:=0.0;
		MDB_Parametros[139]:=0.0;
		MDB_Parametros[140]:=0.0;
//		MDB_Parametros[141]:=VByPass.Parametro.Tempo.Abrir;
//		MDB_Parametros[142]:=VByPass.Parametro.Tempo.Fechar;
		MDB_Parametros[143]:=0.0;
		MDB_Parametros[144]:=0.0;
		MDB_Parametros[145]:=0.0;
		MDB_Parametros[146]:=0.0;
		MDB_Parametros[147]:=0.0;
		MDB_Parametros[148]:=0.0;
		MDB_Parametros[149]:=0.0;
		MDB_Parametros[150]:=0.0;
//		MDB_Parametros[151]:=VBorb.Parametro.Tempo.Abrir;
//		MDB_Parametros[152]:=VBorb.Parametro.Tempo.Fechar;
//		MDB_Parametros[153]:=VBorb.Parametro.Tempo.Equalizar;
//		MDB_Parametros[154]:=VBorb.Parametro.Delta_Pressao;
//		MDB_Parametros[155]:=VBorb.Parametro.Pressao.Montante.SensorMin;
//		MDB_Parametros[156]:=VBorb.Parametro.Pressao.Montante.SensorMax;
//		MDB_Parametros[157]:=VBorb.Parametro.Pressao.Jusante.SensorMin;
//		MDB_Parametros[158]:=VBorb.Parametro.Pressao.Jusante.SensorMax;
		MDB_Parametros[159]:=0.0;
		MDB_Parametros[160]:=0.0;
		MDB_Parametros[161]:=0.0;
		MDB_Parametros[162]:=0.0;
		MDB_Parametros[163]:=0.0;
		MDB_Parametros[164]:=0.0;
		MDB_Parametros[165]:=0.0;
		MDB_Parametros[166]:=0.0;
		MDB_Parametros[167]:=0.0;
		MDB_Parametros[168]:=Comporta1.Parametro.Encoder1_SensorMin;
		MDB_Parametros[169]:=Comporta1.Parametro.Encoder1_SensorMax;
		MDB_Parametros[170]:=Comporta1.Parametro.Tempo_Cracking;
		MDB_Parametros[171]:=Comporta1.Parametro.Tempo_Falha_Abertura;
		MDB_Parametros[172]:=Comporta1.Parametro.Tempo_Falha_Cracking;
		MDB_Parametros[173]:=Comporta1.Parametro.Tempo_Falha_Fechando;
		MDB_Parametros[174]:=Comporta1.Parametro.Tempo_Falha_Reposicao;
//		MDB_Parametros[175]:=Comporta1.Parametro.Pressao.Montante.SensorMin;
//		MDB_Parametros[176]:=Comporta1.Parametro.Pressao.Montante.SensorMax;
		MDB_Parametros[177]:=Comporta2.Parametro.Encoder2_SensorMin;
		MDB_Parametros[178]:=Comporta2.Parametro.Encoder2_SensorMax;
		MDB_Parametros[179]:=Comporta2.Parametro.Tempo_Cracking;
		MDB_Parametros[180]:=Comporta2.Parametro.Tempo_Falha_Abertura;
		MDB_Parametros[181]:=Comporta2.Parametro.Tempo_Falha_Cracking;
		MDB_Parametros[182]:=Comporta2.Parametro.Tempo_Falha_Fechando;
		MDB_Parametros[183]:=Comporta2.Parametro.Tempo_Falha_Reposicao;
		MDB_Parametros[184]:=Comporta_UH.Parametro.Temperatura_Oleo.SensorMin;
		MDB_Parametros[185]:=Comporta_UH.Parametro.Temperatura_Oleo.SensorMax;
		MDB_Parametros[186]:=Comporta_UH.Parametro.Temperatura_Oleo.Alarme;
		MDB_Parametros[187]:=Comporta_UH.Parametro.Temperatura_Oleo.Trip;
		MDB_Parametros[188]:=Comporta_UH.Parametro.Temperatura_Oleo.Tempo_AL;
		MDB_Parametros[189]:=Comporta_UH.Parametro.Temperatura_Oleo.Tempo_TR;
		MDB_Parametros[190]:=0.0;
		MDB_Parametros[191]:=Turbina.Parametro.Gaxeteiro.Temperatura.SensorMin;
		MDB_Parametros[192]:=Turbina.Parametro.Gaxeteiro.Temperatura.SensorMax;
		MDB_Parametros[193]:=Turbina.Parametro.Gaxeteiro.Temperatura.Alarme;
		MDB_Parametros[194]:=Turbina.Parametro.Gaxeteiro.Temperatura.Trip;
		MDB_Parametros[195]:=Turbina.Parametro.Gaxeteiro.Temperatura.Tempo_AL;
		MDB_Parametros[196]:=Turbina.Parametro.Gaxeteiro.Temperatura.Tempo_TR;
		MDB_Parametros[197]:=Turbina.Parametro.Mancal1.Temperatura.SensorMin;
		MDB_Parametros[198]:=Turbina.Parametro.Mancal1.Temperatura.SensorMax;
		MDB_Parametros[199]:=Turbina.Parametro.Mancal1.Temperatura.Alarme;
		MDB_Parametros[200]:=Turbina.Parametro.Mancal1.Temperatura.Trip;
		MDB_Parametros[201]:=Turbina.Parametro.Mancal1.Temperatura.Tempo_AL;
		MDB_Parametros[202]:=Turbina.Parametro.Mancal1.Temperatura.Tempo_TR;
		MDB_Parametros[203]:=Turbina.Parametro.Mancal2.Temperatura.SensorMin;
		MDB_Parametros[204]:=Turbina.Parametro.Mancal2.Temperatura.SensorMax;
		MDB_Parametros[205]:=Turbina.Parametro.Mancal2.Temperatura.Alarme;
		MDB_Parametros[206]:=Turbina.Parametro.Mancal2.Temperatura.Trip;
		MDB_Parametros[207]:=Turbina.Parametro.Mancal2.Temperatura.Tempo_AL;
		MDB_Parametros[208]:=Turbina.Parametro.Mancal2.Temperatura.Tempo_TR;
		MDB_Parametros[209]:=Turbina.Parametro.Mancal3.Temperatura.SensorMin;
		MDB_Parametros[210]:=Turbina.Parametro.Mancal3.Temperatura.SensorMax;
		MDB_Parametros[211]:=Turbina.Parametro.Mancal3.Temperatura.Alarme;
		MDB_Parametros[212]:=Turbina.Parametro.Mancal3.Temperatura.Trip;
		MDB_Parametros[213]:=Turbina.Parametro.Mancal3.Temperatura.Tempo_AL;
		MDB_Parametros[214]:=Turbina.Parametro.Mancal3.Temperatura.Tempo_TR;
		MDB_Parametros[215]:=Turbina.Parametro.Mancal4.Temperatura.SensorMin;
		MDB_Parametros[216]:=Turbina.Parametro.Mancal4.Temperatura.SensorMax;
		MDB_Parametros[217]:=Turbina.Parametro.Mancal4.Temperatura.Alarme;
		MDB_Parametros[218]:=Turbina.Parametro.Mancal4.Temperatura.Trip;
		MDB_Parametros[219]:=Turbina.Parametro.Mancal4.Temperatura.Tempo_AL;
		MDB_Parametros[220]:=Turbina.Parametro.Mancal4.Temperatura.Tempo_TR;
		MDB_Parametros[221]:=Turbina.Parametro.Mancal5.Temperatura.SensorMin;
		MDB_Parametros[222]:=Turbina.Parametro.Mancal5.Temperatura.SensorMax;
		MDB_Parametros[223]:=Turbina.Parametro.Mancal5.Temperatura.Alarme;
		MDB_Parametros[224]:=Turbina.Parametro.Mancal5.Temperatura.Trip;
		MDB_Parametros[225]:=Turbina.Parametro.Mancal5.Temperatura.Tempo_AL;
		MDB_Parametros[226]:=Turbina.Parametro.Mancal5.Temperatura.Tempo_TR;
		MDB_Parametros[227]:=Turbina.Parametro.Mancal6.Temperatura.SensorMin;
		MDB_Parametros[228]:=Turbina.Parametro.Mancal6.Temperatura.SensorMax;
		MDB_Parametros[229]:=Turbina.Parametro.Mancal6.Temperatura.Alarme;
		MDB_Parametros[230]:=Turbina.Parametro.Mancal6.Temperatura.Trip;
		MDB_Parametros[231]:=Turbina.Parametro.Mancal6.Temperatura.Tempo_AL;
		MDB_Parametros[232]:=Turbina.Parametro.Mancal6.Temperatura.Tempo_TR;
		MDB_Parametros[233]:=Turbina.Parametro.CaixaEspiral.Pressao.SensorMin;
		MDB_Parametros[234]:=Turbina.Parametro.CaixaEspiral.Pressao.SensorMax;
		MDB_Parametros[235]:=Turbina.Parametro.CaixaEspiral.Pressao.Alarme;
		MDB_Parametros[236]:=Turbina.Parametro.CaixaEspiral.Pressao.Trip;
		MDB_Parametros[237]:=Turbina.Parametro.CaixaEspiral.Pressao.Tempo_AL;
		MDB_Parametros[238]:=Turbina.Parametro.CaixaEspiral.Pressao.Tempo_TR;
		MDB_Parametros[239]:=Turbina.Parametro.Delta_Pressao;
		MDB_Parametros[240]:=0.0;
		MDB_Parametros[241]:=0.0;
		MDB_Parametros[242]:=0.0;
		MDB_Parametros[243]:=0.0;
		MDB_Parametros[244]:=0.0;
		MDB_Parametros[245]:=0.0;
		MDB_Parametros[246]:=0.0;
		MDB_Parametros[247]:=0.0;
		MDB_Parametros[248]:=0.0;
		MDB_Parametros[249]:=0.0;
		MDB_Parametros[250]:=0.0;
		MDB_Parametros[251]:=Gerador.Parametro.Fase_A.Temperatura.SensorMin;
		MDB_Parametros[252]:=Gerador.Parametro.Fase_A.Temperatura.SensorMax;
		MDB_Parametros[253]:=Gerador.Parametro.Fase_A.Temperatura.Alarme;
		MDB_Parametros[254]:=Gerador.Parametro.Fase_A.Temperatura.Trip;
		MDB_Parametros[255]:=Gerador.Parametro.Fase_A.Temperatura.Tempo_AL;
		MDB_Parametros[256]:=Gerador.Parametro.Fase_A.Temperatura.Tempo_TR;
		MDB_Parametros[257]:=Gerador.Parametro.Fase_B.Temperatura.SensorMin;
		MDB_Parametros[258]:=Gerador.Parametro.Fase_B.Temperatura.SensorMax;
		MDB_Parametros[259]:=Gerador.Parametro.Fase_B.Temperatura.Alarme;
		MDB_Parametros[260]:=Gerador.Parametro.Fase_B.Temperatura.Trip;
		MDB_Parametros[261]:=Gerador.Parametro.Fase_B.Temperatura.Tempo_AL;
		MDB_Parametros[262]:=Gerador.Parametro.Fase_B.Temperatura.Tempo_TR;
		MDB_Parametros[263]:=Gerador.Parametro.Fase_C.Temperatura.SensorMin;
		MDB_Parametros[264]:=Gerador.Parametro.Fase_C.Temperatura.SensorMax;
		MDB_Parametros[265]:=Gerador.Parametro.Fase_C.Temperatura.Alarme;
		MDB_Parametros[266]:=Gerador.Parametro.Fase_C.Temperatura.Trip;
		MDB_Parametros[267]:=Gerador.Parametro.Fase_C.Temperatura.Tempo_AL;
		MDB_Parametros[268]:=Gerador.Parametro.Fase_C.Temperatura.Tempo_TR;
		MDB_Parametros[269]:=Gerador.Parametro.NucleoEstatorico1.Temperatura.SensorMin;
		MDB_Parametros[270]:=Gerador.Parametro.NucleoEstatorico1.Temperatura.SensorMax;
		MDB_Parametros[271]:=Gerador.Parametro.NucleoEstatorico1.Temperatura.Alarme;
		MDB_Parametros[272]:=Gerador.Parametro.NucleoEstatorico1.Temperatura.Trip;
		MDB_Parametros[273]:=Gerador.Parametro.NucleoEstatorico1.Temperatura.Tempo_AL;
		MDB_Parametros[274]:=Gerador.Parametro.NucleoEstatorico1.Temperatura.Tempo_TR;
		MDB_Parametros[275]:=Gerador.Parametro.NucleoEstatorico2.Temperatura.SensorMin;
		MDB_Parametros[276]:=Gerador.Parametro.NucleoEstatorico2.Temperatura.SensorMax;
		MDB_Parametros[277]:=Gerador.Parametro.NucleoEstatorico2.Temperatura.Alarme;
		MDB_Parametros[278]:=Gerador.Parametro.NucleoEstatorico2.Temperatura.Trip;
		MDB_Parametros[279]:=Gerador.Parametro.NucleoEstatorico2.Temperatura.Tempo_AL;
		MDB_Parametros[280]:=Gerador.Parametro.NucleoEstatorico2.Temperatura.Tempo_TR;
		MDB_Parametros[281]:=Gerador.Parametro.NucleoEstatorico3.Temperatura.SensorMin;
		MDB_Parametros[282]:=Gerador.Parametro.NucleoEstatorico3.Temperatura.SensorMax;
		MDB_Parametros[283]:=Gerador.Parametro.NucleoEstatorico3.Temperatura.Alarme;
		MDB_Parametros[284]:=Gerador.Parametro.NucleoEstatorico3.Temperatura.Trip;
		MDB_Parametros[285]:=Gerador.Parametro.NucleoEstatorico3.Temperatura.Tempo_AL;
		MDB_Parametros[286]:=Gerador.Parametro.NucleoEstatorico3.Temperatura.Tempo_TR;
		MDB_Parametros[287]:=Gerador.Parametro.Mancal1.Temperatura.SensorMin;
		MDB_Parametros[288]:=Gerador.Parametro.Mancal1.Temperatura.SensorMax;
		MDB_Parametros[289]:=Gerador.Parametro.Mancal1.Temperatura.Alarme;
		MDB_Parametros[290]:=Gerador.Parametro.Mancal1.Temperatura.Trip;
		MDB_Parametros[291]:=Gerador.Parametro.Mancal1.Temperatura.Tempo_AL;
		MDB_Parametros[292]:=Gerador.Parametro.Mancal1.Temperatura.Tempo_TR;
		MDB_Parametros[293]:=Gerador.Parametro.Mancal2.Temperatura.SensorMin;
		MDB_Parametros[294]:=Gerador.Parametro.Mancal2.Temperatura.SensorMax;
		MDB_Parametros[295]:=Gerador.Parametro.Mancal2.Temperatura.Alarme;
		MDB_Parametros[296]:=Gerador.Parametro.Mancal2.Temperatura.Trip;
		MDB_Parametros[297]:=Gerador.Parametro.Mancal2.Temperatura.Tempo_AL;
		MDB_Parametros[298]:=Gerador.Parametro.Mancal2.Temperatura.Tempo_TR;
		MDB_Parametros[299]:=Gerador.Parametro.Mancal3.Temperatura.SensorMin;
		MDB_Parametros[300]:=Gerador.Parametro.Mancal3.Temperatura.SensorMax;
		MDB_Parametros[301]:=Gerador.Parametro.Mancal3.Temperatura.Alarme;
		MDB_Parametros[302]:=Gerador.Parametro.Mancal3.Temperatura.Trip;
		MDB_Parametros[303]:=Gerador.Parametro.Mancal3.Temperatura.Tempo_AL;
		MDB_Parametros[304]:=Gerador.Parametro.Mancal3.Temperatura.Tempo_TR;
		MDB_Parametros[305]:=Gerador.Parametro.Mancal4.Temperatura.SensorMin;
		MDB_Parametros[306]:=Gerador.Parametro.Mancal4.Temperatura.SensorMax;
		MDB_Parametros[307]:=Gerador.Parametro.Mancal4.Temperatura.Alarme;
		MDB_Parametros[308]:=Gerador.Parametro.Mancal4.Temperatura.Trip;
		MDB_Parametros[309]:=Gerador.Parametro.Mancal4.Temperatura.Tempo_AL;
		MDB_Parametros[310]:=Gerador.Parametro.Mancal4.Temperatura.Tempo_TR;
		MDB_Parametros[311]:=Gerador.Parametro.Mancal5.Temperatura.SensorMin;
		MDB_Parametros[312]:=Gerador.Parametro.Mancal5.Temperatura.SensorMax;
		MDB_Parametros[313]:=Gerador.Parametro.Mancal5.Temperatura.Alarme;
		MDB_Parametros[314]:=Gerador.Parametro.Mancal5.Temperatura.Trip;
		MDB_Parametros[315]:=Gerador.Parametro.Mancal5.Temperatura.Tempo_AL;
		MDB_Parametros[316]:=Gerador.Parametro.Mancal5.Temperatura.Tempo_TR;
		MDB_Parametros[317]:=Gerador.Parametro.Mancal6.Temperatura.SensorMin;
		MDB_Parametros[318]:=Gerador.Parametro.Mancal6.Temperatura.SensorMax;
		MDB_Parametros[319]:=Gerador.Parametro.Mancal6.Temperatura.Alarme;
		MDB_Parametros[320]:=Gerador.Parametro.Mancal6.Temperatura.Trip;
		MDB_Parametros[321]:=Gerador.Parametro.Mancal6.Temperatura.Tempo_AL;
		MDB_Parametros[322]:=Gerador.Parametro.Mancal6.Temperatura.Tempo_TR;
		MDB_Parametros[323]:=0.0;
		MDB_Parametros[324]:=0.0;
		MDB_Parametros[325]:=0.0;
		MDB_Parametros[326]:=0.0;
		MDB_Parametros[327]:=0.0;
		MDB_Parametros[328]:=0.0;
		MDB_Parametros[329]:=0.0;
		MDB_Parametros[330]:=0.0;
		MDB_Parametros[331]:=0.0;
		MDB_Parametros[332]:=0.0;
		MDB_Parametros[333]:=0.0;
		MDB_Parametros[334]:=0.0;
		MDB_Parametros[335]:=0.0;
		MDB_Parametros[336]:=0.0;
		MDB_Parametros[337]:=0.0;
		MDB_Parametros[338]:=0.0;
		MDB_Parametros[339]:=0.0;
		MDB_Parametros[340]:=0.0;
		MDB_Parametros[341]:=RT.Parametro.PWR.Temperatura.SensorMin;
		MDB_Parametros[342]:=RT.Parametro.PWR.Temperatura.SensorMax;
		MDB_Parametros[343]:=RT.Parametro.PWR.Temperatura.Alarme;
		MDB_Parametros[344]:=RT.Parametro.PWR.Temperatura.Trip;
		MDB_Parametros[345]:=RT.Parametro.PWR.Temperatura.Tempo_AL;
		MDB_Parametros[346]:=RT.Parametro.PWR.Temperatura.Tempo_TR;
//		MDB_Parametros[347]:=0.0;
//		MDB_Parametros[348]:=0.0;
//		MDB_Parametros[349]:=0.0;
//		MDB_Parametros[350]:=0.0;
//		MDB_Parametros[351]:=0.0;
//		MDB_Parametros[352]:=0.0;
//		MDB_Parametros[353]:=0.0;
//		MDB_Parametros[354]:=0.0;
//		MDB_Parametros[355]:=0.0;
//		MDB_Parametros[356]:=0.0;
//		MDB_Parametros[357]:=0.0;
//		MDB_Parametros[358]:=0.0;
//		MDB_Parametros[359]:=0.0;
//		MDB_Parametros[360]:=0.0;
		MDB_Parametros[361]:=Trafo_Exc.Parametro.Fase_A.Temperatura.SensorMin;
		MDB_Parametros[362]:=Trafo_Exc.Parametro.Fase_A.Temperatura.SensorMax;
		MDB_Parametros[363]:=Trafo_Exc.Parametro.Fase_A.Temperatura.Alarme;
		MDB_Parametros[364]:=Trafo_Exc.Parametro.Fase_A.Temperatura.Trip;
		MDB_Parametros[365]:=Trafo_Exc.Parametro.Fase_A.Temperatura.Tempo_AL;
		MDB_Parametros[366]:=Trafo_Exc.Parametro.Fase_A.Temperatura.Tempo_TR;
		MDB_Parametros[367]:=Trafo_Exc.Parametro.Fase_B.Temperatura.SensorMin;
		MDB_Parametros[368]:=Trafo_Exc.Parametro.Fase_B.Temperatura.SensorMax;
		MDB_Parametros[369]:=Trafo_Exc.Parametro.Fase_B.Temperatura.Alarme;
		MDB_Parametros[370]:=Trafo_Exc.Parametro.Fase_B.Temperatura.Trip;
		MDB_Parametros[371]:=Trafo_Exc.Parametro.Fase_B.Temperatura.Tempo_AL;
		MDB_Parametros[372]:=Trafo_Exc.Parametro.Fase_B.Temperatura.Tempo_TR;
		MDB_Parametros[373]:=Trafo_Exc.Parametro.Fase_C.Temperatura.SensorMin;
		MDB_Parametros[374]:=Trafo_Exc.Parametro.Fase_C.Temperatura.SensorMax;
		MDB_Parametros[375]:=Trafo_Exc.Parametro.Fase_C.Temperatura.Alarme;
		MDB_Parametros[376]:=Trafo_Exc.Parametro.Fase_C.Temperatura.Trip;
		MDB_Parametros[377]:=Trafo_Exc.Parametro.Fase_C.Temperatura.Tempo_AL;
		MDB_Parametros[378]:=Trafo_Exc.Parametro.Fase_C.Temperatura.Tempo_TR;
//		MDB_Parametros[379]:=0.0;
//		MDB_Parametros[380]:=0.0;
//		MDB_Parametros[381]:=0.0;
//		MDB_Parametros[382]:=0.0;
//		MDB_Parametros[383]:=0.0;
//		MDB_Parametros[384]:=0.0;
//		MDB_Parametros[385]:=0.0;
//		MDB_Parametros[386]:=0.0;
//		MDB_Parametros[387]:=0.0;
//		MDB_Parametros[388]:=0.0;
//		MDB_Parametros[389]:=0.0;
//		MDB_Parametros[390]:=0.0;
		MDB_Parametros[391]:=Nivel.Parametro.Nivel_Ligar;
		MDB_Parametros[392]:=Nivel.Parametro.Nivel_Desligar;
		MDB_Parametros[393]:=Nivel.Parametro.Nivel_Trip;
		MDB_Parametros[394]:=Nivel.Parametro.Nivel_Min;		//Referência
		MDB_Parametros[395]:=Nivel.Parametro.Nivel_Max;		//Não usado
		MDB_Parametros[396]:=Nivel.Parametro.Potencia_Min;
		MDB_Parametros[397]:=Nivel.Parametro.Potencia_Max;
		MDB_Parametros[398]:=Nivel.Parametro.PID.Kp;
		MDB_Parametros[399]:=Nivel.Parametro.PID.Ki;
		MDB_Parametros[400]:=Nivel.Parametro.PID.Kd;
		MDB_Parametros[401]:=Nivel.Parametro.PID.Tf;
		MDB_Parametros[402]:=0.0;
		MDB_Parametros[403]:=0.0;
		MDB_Parametros[404]:=0.0;
		MDB_Parametros[405]:=0.0;
		MDB_Parametros[406]:=0.0;
		MDB_Parametros[407]:=0.0;
		MDB_Parametros[408]:=0.0;
		MDB_Parametros[409]:=0.0;
		MDB_Parametros[410]:=0.0;
		MDB_Parametros[411]:=Nivel.Parametro.Barragem.SensorMin;
		MDB_Parametros[412]:=Nivel.Parametro.Barragem.SensorMax;
		MDB_Parametros[413]:=0.0;
		MDB_Parametros[414]:=0.0;
		MDB_Parametros[415]:=Nivel.Parametro.Barragem.Alarme;
		MDB_Parametros[416]:=Nivel.Parametro.Barragem.Trip;
		MDB_Parametros[417]:=Nivel.Parametro.Barragem.Tempo_AL;
		MDB_Parametros[418]:=Nivel.Parametro.Barragem.Tempo_TR;
		MDB_Parametros[419]:=Nivel.Parametro.Jusante.SensorMin;
		MDB_Parametros[420]:=Nivel.Parametro.Jusante.SensorMax;
		MDB_Parametros[421]:=0.0;
		MDB_Parametros[422]:=Nivel.Parametro.Jusante.Cota;
		MDB_Parametros[423]:=Nivel.Parametro.Jusante.Alarme;
		MDB_Parametros[424]:=Nivel.Parametro.Jusante.Trip;
		MDB_Parametros[425]:=Nivel.Parametro.Jusante.Tempo_AL;
		MDB_Parametros[426]:=Nivel.Parametro.Jusante.Tempo_TR;
		MDB_Parametros[427]:=0.0;
		MDB_Parametros[428]:=0.0;
		MDB_Parametros[429]:=0.0;
		MDB_Parametros[430]:=Nivel.Parametro.Jusante_Grade1.SensorMin;
		MDB_Parametros[431]:=Nivel.Parametro.Jusante_Grade1.SensorMax;
		MDB_Parametros[432]:=Nivel.Parametro.Jusante_Grade1.Cota;
		MDB_Parametros[433]:=Nivel.Parametro.Jusante_Grade1.Alarme;
		MDB_Parametros[434]:=Nivel.Parametro.Jusante_Grade1.Trip;
		MDB_Parametros[435]:=Nivel.Parametro.Jusante_Grade1.Tempo_AL;
		MDB_Parametros[436]:=Nivel.Parametro.Jusante_Grade1.Tempo_TR;
		MDB_Parametros[437]:=0.0;
		MDB_Parametros[438]:=0.0;
		MDB_Parametros[439]:=0.0;
		MDB_Parametros[440]:=Nivel.Parametro.Jusante_Grade2.SensorMin;
		MDB_Parametros[441]:=Nivel.Parametro.Jusante_Grade2.SensorMax;
		MDB_Parametros[442]:=Nivel.Parametro.Jusante_Grade2.Cota;
		MDB_Parametros[443]:=Nivel.Parametro.Jusante_Grade2.Alarme;
		MDB_Parametros[444]:=Nivel.Parametro.Jusante_Grade2.Trip;
		MDB_Parametros[445]:=Nivel.Parametro.Jusante_Grade2.Tempo_AL;
		MDB_Parametros[446]:=Nivel.Parametro.Jusante_Grade2.Tempo_TR;
		MDB_Parametros[447]:=0.0;
		MDB_Parametros[448]:=0.0;
		MDB_Parametros[449]:=0.0;
		MDB_Parametros[450]:=0.0;
		MDB_Parametros[451]:=0.0;
		MDB_Parametros[452]:=0.0;
		MDB_Parametros[453]:=0.0;
		MDB_Parametros[454]:=0.0;
		MDB_Parametros[455]:=0.0;
		MDB_Parametros[456]:=0.0;
		MDB_Parametros[457]:=0.0;
		MDB_Parametros[458]:=0.0;
		MDB_Parametros[459]:=0.0;
		MDB_Parametros[460]:=0.0;

	//-------------------------------------------------------------------------------------------
	END_IF;

	//-------------------------------------------------------------------------------------------
	(*Nível Camara de Carga*)
	IF link_MDB_Nv_CC.NewValue THEN
		link_MDB_Nv_CC.NewValue    := FALSE;

		Painel.PSA.Medidas.Nivel_Barragem	:= Painel.PSA.Rede.NIVEL_BARRAGEM;
	END_IF;

END_PROGRAM
```

### Program Logical/Auto/Modbus/MDB_STS

#### Cyclic.st
```iecst
PROGRAM _CYCLIC

 	//-------------------------------------------------------------------------------------------
	(*Status*)
	//-------------------------------------------------------------------------------------------

	MDB_Status[1] := UG.Status.Motivo_Parada_Normal;
	MDB_Status[2] := UG.Status.Motivo_Parada_86M;
	MDB_Status[3] := UG.Status.Motivo_Parada_86E;
	MDB_Status[4] := UG.Status.Motivo_Parada_86H;
	MDB_Status[5] := UG.Status.Motivo_Parada_Nivel;
	MDB_Status[6] := UG.Status.Automatico;
	MDB_Status[7] := UG.Status.Manual;
	MDB_Status[8] := UG.Status.Manutencao;
	MDB_Status[9] := UG.Status.UP_Partindo;
	MDB_Status[10] := UG.Status.UP_Alvo;
	MDB_Status[11] := UG.Status.UP;
	MDB_Status[12] := UG.Status.UPGM_Precond;
	MDB_Status[13] := UG.Status.UPGM_Partindo;
	MDB_Status[14] := UG.Status.UPGM_Parando;
	MDB_Status[15] := UG.Status.UPGM_Alvo;
	MDB_Status[16] := UG.Status.UPGM;
	MDB_Status[17] := UG.Status.UMVD_Precond;
	MDB_Status[18] := UG.Status.UMVD_Partindo;
	MDB_Status[19] := UG.Status.UMVD_Parando;
	MDB_Status[20] := UG.Status.UMVD_Alvo;
	MDB_Status[21] := UG.Status.UMVD;
	MDB_Status[22] := UG.Status.UPS_Precond;
	MDB_Status[23] := UG.Status.UPS_Partindo;
	MDB_Status[24] := UG.Status.UPS_Parando;
	MDB_Status[25] := UG.Status.UPS_Alvo;
	MDB_Status[26] := UG.Status.UPS;
	MDB_Status[27] := UG.Status.US_Precond;
	MDB_Status[28] := UG.Status.US_Parando;
	MDB_Status[29] := UG.Status.US_Alvo;
	MDB_Status[30] := UG.Status.US;
	MDB_Status[31] := FALSE;
	MDB_Status[32] := FALSE;
	MDB_Status[33] := FALSE;
	MDB_Status[34] := FALSE;
	MDB_Status[35] := FALSE;
	MDB_Status[36] := FALSE;
	MDB_Status[37] := FALSE;
	MDB_Status[38] := FALSE;
	MDB_Status[39] := FALSE;
	MDB_Status[40] := FALSE;
	MDB_Status[41] := Painel.Status.Rele_86;
	MDB_Status[42] := Painel.Status.Rele_86E;
	MDB_Status[43] := Painel.Status.Rele_86M;
	MDB_Status[44] := Painel.Status.Rele_86H;
	MDB_Status[45] := Painel.Status.Local;
	MDB_Status[46] := Painel.Status.Remoto;
	MDB_Status[47] := Painel.Status.Reset;
	MDB_Status[48] := FALSE;
	MDB_Status[49] := FALSE;
	MDB_Status[50] := FALSE;
	MDB_Status[51] := FALSE;
	MDB_Status[52] := FALSE;
	MDB_Status[53] := FALSE;
	MDB_Status[54] := FALSE;
	MDB_Status[55] := FALSE;
	MDB_Status[56] := FALSE;
	MDB_Status[57] := FALSE;
	MDB_Status[58] := FALSE;
	MDB_Status[59] := FALSE;
	MDB_Status[60] := SFA.Status.Habilitado;
	MDB_Status[61] := SFA.Status.Bomba1.Ligado;
	MDB_Status[62] := SFA.Status.Bomba1.Desligado;
	MDB_Status[63] := FALSE;
	MDB_Status[64] := FALSE;
	MDB_Status[65] := SFA.Status.Filtro1_Valv_Entrada1.Aberto;
	MDB_Status[66] := SFA.Status.Filtro1_Valv_Retrolav1.Aberto;
	MDB_Status[67] := SFA.Status.Filtro1_Valv_Entrada2.Aberto;
	MDB_Status[68] := SFA.Status.Filtro1_Valv_Retrolav2.Aberto;
	MDB_Status[69] := SFA.Status.Filtro2_Valv_Entrada1.Aberto;
	MDB_Status[70] := SFA.Status.Filtro2_Valv_Retrolav1.Aberto;
	MDB_Status[71] := SFA.Status.Filtro2_Valv_Entrada2.Aberto;
	MDB_Status[72] := SFA.Status.Filtro2_Valv_Retrolav2.Aberto;
	MDB_Status[73] := SFA.Status.Pressao.Normal;
	MDB_Status[74] := FALSE;
	MDB_Status[75] := FALSE;
	MDB_Status[76] := FALSE;
	MDB_Status[77] := FALSE;
	MDB_Status[78] := FALSE;
	MDB_Status[79] := FALSE;
	MDB_Status[80] := FALSE;
	MDB_Status[81] := UHLM.Status.Habilitado;
	MDB_Status[82] := UHLM.Status.Desabilitado;
	MDB_Status[83] := UHLM.Status.Local;
	MDB_Status[84] := UHLM.Status.Remoto;
	MDB_Status[85] := UHLM.Status.Partindo;
	MDB_Status[86] := UHLM.Status.Parando;
	MDB_Status[87] := UHLM.Status.Bomba1.Ligado;
	MDB_Status[88] := UHLM.Status.Bomba1.Desligado;
	MDB_Status[89] := UHLM.Status.Bomba2.Ligado;
	MDB_Status[90] := UHLM.Status.Bomba2.Desligado;
	MDB_Status[91] := UHLM.Status.JackingOil.Ligado;
	MDB_Status[92] := UHLM.Status.JackingOil.Desligado;
	MDB_Status[93] := UHLM.Status.Ventilador.Ligado;
	MDB_Status[94] := UHLM.Status.Ventilador.Desligado;
	MDB_Status[95] := UHLM.Status.Nivel.Normal;
	MDB_Status[96] := UHLM.Status.Temperatura.Normal;
	MDB_Status[97] := UHLM.Status.Fluxo.Normal;
	MDB_Status[98] := UHLM.Status.Fluxo1.Normal;(*Fluxostato do trocador de calor do mancal combinado*)
	MDB_Status[99] := UHLM.Status.Fluxo2.Normal;(*Fluxostato do trocador de calor do mancal guia*)
	MDB_Status[100] := UHLM.Status.Fluxo3.Normal;
	MDB_Status[101] := UHLM.Status.Fluxo4.Normal;
	MDB_Status[102] := UHLM.Status.Fluxo5.Normal;
	MDB_Status[103] := UHLM.Status.Pressao.Normal;
	MDB_Status[104] := UHLM.Status.Pressao1.Normal;(*Pressostato da linha de óleo jacking oil*)
	MDB_Status[105] := UHLM.Status.Pressao2.Normal;(*Pressostato da linha de óleo mancal combinado*)
	MDB_Status[106] := UHLM.Status.Pressao3.Normal;(*Pressostato da linha de óleo mancal guia*)
	MDB_Status[107] := UHLM.Status.Pressao4.Normal;
	MDB_Status[108] := UHLM.Status.Pressao5.Normal;
	MDB_Status[109] := UHLM.Status.Bomba3.Ligado;
	MDB_Status[110] := UHLM.Status.Bomba3.Desligado;
	MDB_Status[111] := UHLM.Status.Nivel_Mancal_Guia.Normal;
	MDB_Status[112] := FALSE;
	MDB_Status[113] := FALSE;
	MDB_Status[114] := FALSE;
	MDB_Status[115] := FALSE;
	MDB_Status[116] := FALSE;
	MDB_Status[117] := FALSE;
	MDB_Status[118] := FALSE;
	MDB_Status[119] := FALSE;
	MDB_Status[120] := FALSE;
	MDB_Status[121] := UHRV.Status.Habilitado;
	MDB_Status[122] := UHRV.Status.Desabilitado;
	MDB_Status[123] := UHRV.Status.Local;
	MDB_Status[124] := UHRV.Status.Remoto;
	MDB_Status[125] := UHRV.Status.Partindo;
	MDB_Status[126] := UHRV.Status.Parando;
	MDB_Status[127] := UHRV.Status.Bomba1.Ligado;
	MDB_Status[128] := UHRV.Status.Bomba1.Desligado;
	MDB_Status[129] := UHRV.Status.Bomba2.Ligado;
	MDB_Status[130] := UHRV.Status.Bomba2.Desligado;
	MDB_Status[131] := UHRV.Status.Bomba3.Ligado;
	MDB_Status[132] := UHRV.Status.Bomba3.Desligado;
	MDB_Status[133] := UHRV.Status.Ventilador.Ligado;
	MDB_Status[134] := UHRV.Status.Ventilador.Desligado;
	MDB_Status[135] := UHRV.Status.Vseg1.Ligado;
	MDB_Status[136] := UHRV.Status.Vseg1.Desligado;
	MDB_Status[137] := UHRV.Status.Vseg2.Ligado;
	MDB_Status[138] := UHRV.Status.Vseg2.Desligado;
	MDB_Status[139] := UHRV.Status.Ventagem.Ligado;
	MDB_Status[140] := UHRV.Status.Ventagem.Desligado;
	MDB_Status[141] := UHRV.Status.Nivel.Normal;
	MDB_Status[142] := UHRV.Status.Temperatura.Normal;
	MDB_Status[143] := UHRV.Status.Pressao.Normal;
	MDB_Status[144] := UHRV.Status.Filtro1.Pressao.Normal;
	MDB_Status[145] := FALSE;
	MDB_Status[146] := FALSE;
	MDB_Status[147] := FALSE;
	MDB_Status[148] := FALSE;
	MDB_Status[149] := FALSE;
	MDB_Status[150] := FALSE;
	MDB_Status[151] := FALSE;
	MDB_Status[152] := FALSE;
	MDB_Status[153] := FALSE;
	MDB_Status[154] := FALSE;
	MDB_Status[155] := FALSE;
	MDB_Status[156] := FALSE;
	MDB_Status[157] := FALSE;
	MDB_Status[158] := FALSE;
	MDB_Status[159] := FALSE;
	MDB_Status[160] := FALSE;
	MDB_Status[161] := Freio.Status.Modo_Continuo;
	MDB_Status[162] := Freio.Status.Modo_Intermitente;
	MDB_Status[163] := Freio.Status.Aplicado;
	MDB_Status[164] := Freio.Status.Desaplicado;
	MDB_Status[165] := Freio.Status.Pressostato_OK;
	MDB_Status[166] := FALSE;
	MDB_Status[167] := FALSE;
	MDB_Status[168] := FALSE;
	MDB_Status[169] := FALSE;
	MDB_Status[170] := FALSE;
//	MDB_Status[171] := VByPass.Status.Aberto;
//	MDB_Status[172] := VByPass.Status.Fechado;
//	MDB_Status[173] := VByPass.Status.Abrindo;
//	MDB_Status[174] := VByPass.Status.Fechando;
	MDB_Status[175] := FALSE;
	MDB_Status[176] := FALSE;
	MDB_Status[177] := FALSE;
	MDB_Status[178] := FALSE;
	MDB_Status[179] := FALSE;
	MDB_Status[180] := FALSE;
	MDB_Status[181] := FALSE;
	MDB_Status[182] := FALSE;
	MDB_Status[183] := FALSE;
	MDB_Status[184] := FALSE;
	MDB_Status[185] := FALSE;
	MDB_Status[186] := FALSE;
	MDB_Status[187] := FALSE;
	MDB_Status[188] := FALSE;
	MDB_Status[189] := FALSE;
	MDB_Status[190] := FALSE;
//	MDB_Status[191] := VBorb.Status.Aberto;
//	MDB_Status[192] := VBorb.Status.Fechado;
//	MDB_Status[193] := VBorb.Status.Abrindo;
//	MDB_Status[194] := VBorb.Status.Fechando;
//	MDB_Status[195] := VBorb.Status.Equalizado;
//	MDB_Status[196] := VBorb.Status.Reposicao;
//	MDB_Status[197] := VBorb.Status.Deriva;
	MDB_Status[198] := FALSE;
	MDB_Status[199] := FALSE;
	MDB_Status[200] := FALSE;
	MDB_Status[201] := FALSE;
	MDB_Status[202] := FALSE;
	MDB_Status[203] := FALSE;
	MDB_Status[204] := FALSE;
	MDB_Status[205] := FALSE;
	MDB_Status[206] := FALSE;
	MDB_Status[207] := FALSE;
	MDB_Status[208] := FALSE;
	MDB_Status[209] := FALSE;
	MDB_Status[210] := FALSE;
	MDB_Status[211] := Comporta1.Status.Aberto;
	MDB_Status[212] := Comporta1.Status.Fechado;
	MDB_Status[213] := Comporta1.Status.Abrindo;
	MDB_Status[214] := Comporta1.Status.Fechando;
	MDB_Status[215] := Comporta1.Status.Cracking;
	MDB_Status[216] := Comporta1.Status.Deriva;
	MDB_Status[217] := Comporta1.Status.Reposicao;
	MDB_Status[218] := FALSE;
	MDB_Status[219] := Comporta2.Status.Aberto;
	MDB_Status[220] := Comporta2.Status.Fechado;
	MDB_Status[221] := Comporta2.Status.Abrindo;
	MDB_Status[222] := Comporta2.Status.Fechando;
	MDB_Status[223] := Comporta2.Status.Cracking;
	MDB_Status[224] := Comporta2.Status.Deriva;
	MDB_Status[225] := Comporta2.Status.Reposicao;
	MDB_Status[226] := Comporta_UH.Status.Bomba1.Ligado;
	MDB_Status[227] := Comporta_UH.Status.Bomba2.Ligado;
	MDB_Status[228] := Comporta_UH.Status.Valv_Abertura_Lenta.Ligado;
	MDB_Status[229] := Comporta_UH.Status.Val_Abertura.Ligado;
	MDB_Status[230] := Comporta_UH.Status.Val_Fechamento.Ligado;
	MDB_Status[231] := Comporta_UH.Status.Valv_Fechamento_Rapido.Ligado;
	MDB_Status[232] := Comportas.Status.Modo_Remoto;
	MDB_Status[233] := Comportas.Status.Pressao_Equalizada;
	MDB_Status[234] := FALSE;
	MDB_Status[235] := FALSE;
	MDB_Status[236] := FALSE;
	MDB_Status[237] := FALSE;
	MDB_Status[238] := FALSE;
	MDB_Status[239] := FALSE;
	MDB_Status[240] := FALSE;
	MDB_Status[241] := RV.Status.Habilitado;
	MDB_Status[242] := RV.Status.Desabilitado;
	MDB_Status[243] := RV.Status.Partindo;
	MDB_Status[244] := RV.Status.Parando;
	MDB_Status[245] := RV.Status.Carga_Zerada;
	MDB_Status[246] := RV.Status.Velocidade_Nominal;
	MDB_Status[247] := RV.Status.Velocidade_30;
	MDB_Status[248] := RV.Status.Velocidade_Parado;
	MDB_Status[249] := FALSE;
	MDB_Status[250] := FALSE;
	MDB_Status[251] := FALSE;
	MDB_Status[252] := FALSE;
	MDB_Status[253] := FALSE;
	MDB_Status[254] := FALSE;
	MDB_Status[255] := FALSE;
	MDB_Status[256] := FALSE;
	MDB_Status[257] := FALSE;
	MDB_Status[258] := FALSE;
	MDB_Status[259] := FALSE;
	MDB_Status[260] := FALSE;
	MDB_Status[261] := RT.Status.Habilitado;
	MDB_Status[262] := RT.Status.Desabilitado;
	MDB_Status[263] := RT.Status.Partindo;
	MDB_Status[264] := RT.Status.Parando;
	MDB_Status[265] := RT.Status.Qm_Constante;
	MDB_Status[266] := RT.Status.FP_Constante;
	MDB_Status[267] := RT.Status.Tensao_Nominal;
	MDB_Status[268] := FALSE;
	MDB_Status[269] := FALSE;
	MDB_Status[270] := FALSE;
	MDB_Status[271] := FALSE;
	MDB_Status[272] := FALSE;
	MDB_Status[273] := FALSE;
	MDB_Status[274] := FALSE;
	MDB_Status[275] := FALSE;
	MDB_Status[276] := FALSE;
	MDB_Status[277] := FALSE;
	MDB_Status[278] := FALSE;
	MDB_Status[279] := FALSE;
	MDB_Status[280] := FALSE;
	MDB_Status[281] := SC.Status.Habilitado;
	MDB_Status[282] := SC.Status.Desabilitado;
	MDB_Status[283] := FALSE;
	MDB_Status[284] := FALSE;
	MDB_Status[285] := FALSE;
	MDB_Status[286] := FALSE;
	MDB_Status[287] := FALSE;
	MDB_Status[288] := FALSE;
	MDB_Status[289] := FALSE;
	MDB_Status[290] := FALSE;
	MDB_Status[291] := DJ52G.Status.Aberto;
	MDB_Status[292] := DJ52G.Status.Fechado;
	MDB_Status[293] := DJ52G.Status.Mola_Carregada;
	MDB_Status[294] := DJ52G.Status.Bobina_Minima;
	MDB_Status[295] := DJ52G.Status.Modo_Teste;
	MDB_Status[296] := DJ52G.Status.Inserido;
	MDB_Status[297] := DJ52G.Status.Extraido;
	MDB_Status[298] := DJ52G.Status.Habilitado;
	MDB_Status[299] := DJ52G.Status.Desabilitado;
	MDB_Status[300] := FALSE;
	MDB_Status[301] := FALSE;
	MDB_Status[302] := FALSE;
	MDB_Status[303] := FALSE;
	MDB_Status[304] := FALSE;
	MDB_Status[305] := FALSE;
	MDB_Status[306] := FALSE;
	MDB_Status[307] := FALSE;
	MDB_Status[308] := FALSE;
	MDB_Status[309] := FALSE;
	MDB_Status[310] := FALSE;
//	MDB_Status[311] := DJ52L.Status.Aberto;
//	MDB_Status[312] := DJ52L.Status.Fechado;
//	MDB_Status[313] := DJ52L.Status.Remoto;
//	MDB_Status[314] := DJ52L.Status.Bloqueio;
	MDB_Status[315] := FALSE;
	MDB_Status[316] := FALSE;
	MDB_Status[317] := FALSE;
	MDB_Status[318] := FALSE;
	MDB_Status[319] := FALSE;
	MDB_Status[320] := FALSE;
	MDB_Status[321] := Nivel.Status.Habilitado;
	MDB_Status[322] := Nivel.Status.Desabilitado;
	MDB_Status[323] := Nivel.Status.Partindo;
	MDB_Status[324] := Nivel.Status.Parando;
	MDB_Status[325] := FALSE;
	MDB_Status[326] := FALSE;
	MDB_Status[327] := FALSE;
	MDB_Status[328] := FALSE;
	MDB_Status[329] := FALSE;
	MDB_Status[330] := FALSE;

	//-------------------------------------------------------------------------------------------
END_PROGRAM
```

### Share.var
```iecst
VAR
	UfAvg : REAL;
	IfAvg : REAL;
END_VAR
```

- Share.var.bak (not shown)

- Cyclic.st.bak (not shown)

- Init.st.bak (not shown)

- Variables.var.bak (not shown)

- Share.typ.bak (not shown)

- Share.var.bak (not shown)

### Program Logical/Kontrol/Hardware/Hardware

#### Variables.var
```iecst
VAR
	Update0985 : BOOL;
	(*UpdateAI4622 : BOOL;
	UpdateAO4622 : BOOL;*)
	reset_cfg_net : TON;
END_VAR
```

- Cyclic.st.bak (not shown)

#### Init.st
```iecst
PROGRAM _INIT
    TagManager(enable:=TRUE);

    //Config Network
    CfgNet.enable   := TRUE;
    PgsCfgNetRegister(TagManager.ident, CfgNet);

    //CM0985
    cm0985.pDeviceName			:= ADR('IF6.ST1');
    cm0985();
    //Link child blocks
    cm0985Gen.Ident				:= cm0985.Ident;
    cm0985Main.Ident			:= cm0985.Ident;
    cm0985Bus.Ident				:= cm0985.Ident;
    cm0985Sync.Ident			:= cm0985.Ident;
    cm0985GenPu.Ident			:= cm0985.Ident;
    cm0985GenPf.Ident			:= cm0985.Ident;
    cm0985GenPa.Ident			:= cm0985.Ident;
    cm0985GenPc.Ident			:= cm0985.Ident;
    cm0985GenPp.Ident           := cm0985.Ident;
    cm0985DO1.Ident				:= cm0985.Ident;
    cm0985Update.Ident			:= cm0985.Ident;
    cm0985Meter.Ident			:= cm0985.Ident;
    //Update Module CM0985
    Update0985  := TRUE;

    //Register Parameters
    PgsTagStartNode     (TagManager.ident, ADR('hwr'));
    //CM0985 Module
    PgsTagStartNode     (TagManager.ident, ADR('cm0985'));
    //CM0985 - CPU
    //    PgsTagRegisterBOOL  (TagManager.ident, TRUE, ADR('ClockWise'),      cm0985.ClockWise);
    PgsTagRegisterBOOL  (TagManager.ident, TRUE, ADR('EnableSetDO5'),   cm0985.EnableSetDO5);
    PgsTagRegisterBOOL  (TagManager.ident, TRUE, ADR('EnableSetDO6'),   cm0985.EnableSetDO6);
    //CM0985 - X2 and X3 - Generator
    PgsTagStartNode     (TagManager.ident, ADR('gen'));
    //    PgsTagRegisterENUM  (TagManager.ident, TRUE, ADR('Connection'),     ADR(cm0985Gen.Connection));
    //    PgsTagRegisterREAL  (TagManager.ident, TRUE, ADR('Vprim'),          cm0985Gen.Vprim);
    //    PgsTagRegisterREAL  (TagManager.ident, TRUE, ADR('Vsec'),           cm0985Gen.Vsec);
    //    PgsTagRegisterREAL  (TagManager.ident, TRUE, ADR('Vnom'),           cm0985Gen.Vnom);
    //    PgsTagRegisterREAL  (TagManager.ident, TRUE, ADR('Iprim'),          cm0985Gen.Iprim);
    //    PgsTagRegisterUSINT (TagManager.ident, TRUE, ADR('Isec'),           cm0985Gen.Isec);
    //    PgsTagRegisterREAL  (TagManager.ident, TRUE, ADR('Inom'),           cm0985Gen.Inom);
    PgsTagRegisterBOOL  (TagManager.ident, TRUE, ADR('EnableHarmonic'), cm0985Gen.EnableHarmonic);
    PgsTagRegisterUINT  (TagManager.ident, TRUE, ADR('Tfilter'),        cm0985Gen.Tfilter);
    PgsTagRegisterREAL  (TagManager.ident, TRUE, ADR('D02Pulse'),       cm0985Gen.D02Pulse);
    PgsTagEndNode       (TagManager.ident);//gen
    //CM0985 - X4 and X6 - Main
    PgsTagStartNode     (TagManager.ident, ADR('main'));
    //    PgsTagRegisterBOOL  (TagManager.ident, TRUE, ADR('Enable3phase'),   cm0985Main.Enable3phase);
    //    PgsTagRegisterENUM  (TagManager.ident, TRUE, ADR('Connection1'),    ADR(cm0985Main.Connection1));
    //    PgsTagRegisterREAL  (TagManager.ident, TRUE, ADR('V1prim'),         cm0985Main.V1prim);
    //    PgsTagRegisterREAL  (TagManager.ident, TRUE, ADR('V1sec'),          cm0985Main.V1sec);
    //    PgsTagRegisterREAL  (TagManager.ident, TRUE, ADR('V1nom'),          cm0985Main.V1nom);
    PgsTagRegisterENUM  (TagManager.ident, TRUE, ADR('Connection2'),    ADR(cm0985Main.Connection2));
    PgsTagRegisterREAL  (TagManager.ident, TRUE, ADR('V2prim'),         cm0985Main.V2prim);
    PgsTagRegisterREAL  (TagManager.ident, TRUE, ADR('V2sec'),          cm0985Main.V2sec);
    PgsTagRegisterREAL  (TagManager.ident, TRUE, ADR('V2nom'),          cm0985Main.V2nom);
    PgsTagEndNode       (TagManager.ident);//main
    //CM0985 - X5 - Bus
    PgsTagStartNode     (TagManager.ident, ADR('bus'));
    PgsTagRegisterENUM  (TagManager.ident, TRUE, ADR('Connection'),     ADR(cm0985Bus.Connection));
    //    PgsTagRegisterREAL  (TagManager.ident, TRUE, ADR('Vprim'),          cm0985Bus.Vprim);
    //    PgsTagRegisterREAL  (TagManager.ident, TRUE, ADR('Vsec'),           cm0985Bus.Vsec);
    //    PgsTagRegisterREAL  (TagManager.ident, TRUE, ADR('Vnom'),           cm0985Bus.Vnom);
    PgsTagEndNode       (TagManager.ident);//bus
    //CM0985 - Sync
    PgsTagStartNode     (TagManager.ident, ADR('sync'));
    PgsTagRegisterENUM  (TagManager.ident, TRUE, ADR('Mode'),           ADR(cm0985Sync.Mode));
    PgsTagRegisterBOOL  (TagManager.ident, TRUE, ADR('ChangeDO4toDo6'), cm0985Sync.ChangeDO4toDo6);
    //    PgsTagRegisterREAL  (TagManager.ident, TRUE, ADR('dFmax'),          cm0985Sync.dFmax);
    //    PgsTagRegisterREAL  (TagManager.ident, TRUE, ADR('dFmin'),          cm0985Sync.dFmin);
    //    PgsTagRegisterREAL  (TagManager.ident, TRUE, ADR('dUmax'),          cm0985Sync.dUmax);
    //    PgsTagRegisterREAL  (TagManager.ident, TRUE, ADR('dAngleMax'),      cm0985Sync.dAngleMax);
    //    PgsTagRegisterREAL  (TagManager.ident, TRUE, ADR('PhaseShift'),     cm0985Sync.PhaseShift);
    PgsTagRegisterREAL  (TagManager.ident, TRUE, ADR('UBmin'),          cm0985Sync.UBmin);
    PgsTagRegisterREAL  (TagManager.ident, TRUE, ADR('DO4Pulse'),       cm0985Sync.DO4Pulse);
    PgsTagRegisterREAL  (TagManager.ident, TRUE, ADR('DO4SwTime'),      cm0985Sync.DO4SwTime);
    PgsTagRegisterREAL  (TagManager.ident, TRUE, ADR('DO6Pulse'),       cm0985Sync.DO6Pulse);
    PgsTagRegisterREAL  (TagManager.ident, TRUE, ADR('DO6SwTime'),      cm0985Sync.DO6SwTime);
    PgsTagEndNode       (TagManager.ident);//sync
    PgsTagEndNode       (TagManager.ident);//cm0985
    PgsTagEndNode       (TagManager.ident);//hwr

END_PROGRAM
```

- Init.st.bak (not shown)

- Variables.var.bak (not shown)

### Share.typ
```iecst
TYPE
	PgsSysParType : 	STRUCT
		Sync : PgsSyncParType;
		Exc : PgsExcParType;
		Gen : PgsGenParType;
	END_STRUCT;
	PgsSyncParType : 	STRUCT
		U1Prim : REAL; (*Volts*)
		U1Sec : REAL; (*Volts*)
		Enable3Phase : REAL;
		Connection : REAL;
		U1Nom : REAL; (*Volts*)
		UBmin : REAL;
		dFmax : REAL; (*Hz*)
		dFmin : REAL; (*Hz*)
		dUmax : REAL; (*%*)
		dAngleMax : REAL; (*Degrees*)
		PhaseShift : REAL; (*Degrees*)
	END_STRUCT;
	PgsExcParType : 	STRUCT
		UexcPrim : REAL; (*Volts*)
		UexcSec : REAL; (*Volts*)
		UexcNom : REAL; (*Volts*)
	END_STRUCT;
	PgsGenParType : 	STRUCT
		UmPrim : REAL; (*Volts*)
		UmSec : REAL; (*Volts*)
		ImPrim : REAL; (*Amper*)
		ImSec : REAL; (*Amper*)
		UmNom : REAL; (*Volts*)
		SmNom : REAL; (*kW*)
		FmNom : REAL; (*Hz*)
		UfMin : REAL; (*Vcc*)
		UfMax : REAL; (*Vcc*)
		UfNom : REAL; (*Volts*)
		IfMin : REAL; (*Acc*)
		IfMax : REAL; (*Acc*)
		IfNom : REAL; (*Amper*)
		RpmNom : REAL; (*RPM*)
		PPR1 : REAL; (*Pulse Per Revolution*)
		Pos1_0p : REAL; (*mA or V*)
		Pos1_100p : REAL; (*mA or V*)
		Pos2_0p : REAL; (*mA or V*)
		Pos2_100p : REAL; (*mA or V*)
		Pos3_0p : REAL; (*mA or V*)
		Pos3_100p : REAL; (*mA or V*)
		ClockWise : REAL;
		Connection : REAL;
		dRpm1Max : REAL; (*RPM/s*)
		PPR2 : REAL; (*Pulse Per Revolution*)
		dRpm2Max : REAL; (*RPM/s*)
	END_STRUCT;
	PgsSysUpdateType : 	STRUCT
		UpdateGen : BOOL;
		UpdateSync : BOOL;
		UpdateBus : BOOL;
		UpdateProt : BOOL;
		ResetRunningHourMeter : BOOL;
		ResetOnlineHourMeter : BOOL;
		ResetEnergy : BOOL;
		EnableSync : BOOL;
		EnableDeadBus : BOOL;
		reserv6 : BOOL;
		reserv7 : BOOL;
		UpdateIO : BOOL;
		reserv9 : BOOL;
		reserv10 : BOOL;
		reserv11 : BOOL;
		RestoreAll : BOOL;
		SaveAll : BOOL;
		UpdateAll : BOOL;
		var1 : BOOL;
		var2 : BOOL;
		var3 : BOOL;
		var4 : BOOL;
		var5 : BOOL;
		var6 : BOOL;
		var7 : BOOL;
		var8 : BOOL;
		var9 : BOOL;
		var10 : BOOL;
		var11 : BOOL;
		var12 : BOOL;
		var13 : BOOL;
		var14 : BOOL;
		var15 : BOOL;
		var16 : BOOL;
		var17 : BOOL;
		var18 : BOOL;
		var19 : BOOL;
		var20 : BOOL;
		var21 : BOOL;
		var22 : BOOL;
		var23 : BOOL;
		var24 : BOOL;
		var25 : BOOL;
		var26 : BOOL;
		var27 : BOOL;
		var28 : BOOL;
		var29 : BOOL;
		var30 : BOOL;
		var31 : BOOL;
		var32 : BOOL;
	END_STRUCT;
	PgsIOParType : 	STRUCT
		AI1Type : REAL;
		AI2Type : REAL;
		AI3Type : REAL;
		AI4Type : REAL;
		AO1Type : REAL;
		AO2Type : REAL;
		AO3Type : REAL;
		AO4Type : REAL;
		AO1min : REAL; (*Analog Output % => Minumum Control*)
		AO1max : REAL; (*Analog Output % => Maximum Control*)
		AO2min : REAL; (*Analog Output % => Minumum Control*)
		AO2max : REAL; (*Analog Output % => Maximum Control*)
		AO3min : REAL; (*Analog Output % => Minumum Control*)
		AO3max : REAL; (*Analog Output % => Maximum Control*)
		AO4min : REAL; (*Analog Output % => Minumum Control*)
		AO4max : REAL; (*Analog Output % => Maximum Control*)
	END_STRUCT;
END_TYPE
```

### Share.var
```iecst
(*System Parameters*)
VAR
	SysPar : PgsSysParType := (Sync:=(U1Prim:=115,U1Sec:=115,Enable3Phase:=0,Connection:=0,U1Nom:=115,UBmin:=0.05,dFmax:=0.3,dFmin:=-0.3,dUmax:=10,dAngleMax:=5,PhaseShift:=0),Exc:=(UexcPrim:=80,UexcSec:=80,UexcNom:=80),Gen:=(UmPrim:=380,UmSec:=380,ImPrim:=800,ImSec:=5,UmNom:=380,SmNom:=500,FmNom:=60,UfMin:=0,UfMax:=150,UfNom:=100,IfMin:=0,IfMax:=20,IfNom:=10,RpmNom:=2000,PPR1:=500,Pos1_0p:=4,Pos1_100p:=20,Pos2_0p:=4,Pos2_100p:=20,Pos3_0p:=4,Pos3_100p:=20,ClockWise:=1,Connection:=0,dRpm1Max:=50,PPR2:=500,dRpm2Max:=50));
	SysUpdate : PgsSysUpdateType;
	SysIOPar : PgsIOParType := (AI1Type:=2,AI2Type:=2,AI3Type:=2,AI4Type:=2,AO1Type:=1,AO2Type:=2,AO3Type:=2,AO4Type:=2,AO1min:=0,AO1max:=100,AO2min:=0,AO2max:=100,AO3min:=0,AO3max:=100,AO4min:=0,AO4max:=100);
	MdbMeter : ARRAY[0..100] OF REAL;
END_VAR
```

### Program Logical/Kontrol/System/System

#### Cyclic.st
```iecst
PROGRAM _CYCLIC

	IF SysUpdate.SaveAll THEN
		SysUpdate.SaveAll		:= FALSE;
		SysUpdate.UpdateAll     := TRUE;
		TagUpdate.write         := TRUE;
	END_IF;

	IF PgsTagValid(TagManager.ident) AND SysUpdate.UpdateAll THEN
		SysUpdate.UpdateAll		:= FALSE;
		SysUpdate.UpdateGen		:= TRUE;
		SysUpdate.UpdateSync	:= TRUE;
		SysUpdate.UpdateBus		:= TRUE;
		SysUpdate.UpdateProt	:= TRUE;
		SysUpdate.UpdateIO      := TRUE;

		avr.Update				:= TRUE;
		gov.Update				:= TRUE;
		pos1.Update				:= TRUE;
		pos2.Update				:= TRUE;
		pos3.Update				:= TRUE;
	END_IF;

	IF SysUpdate.UpdateGen THEN
		SysUpdate.UpdateGen         := FALSE;
		SysUpdate.UpdateProt		:= TRUE;

		//Meter Base
		meter.Base.Um               := SysPar.Gen.UmNom;
		meter.Base.Sm               := SysPar.Gen.SmNom;
		meter.Base.Rot              := SysPar.Gen.RpmNom;
		meter.Base.Fm               := SysPar.Gen.FmNom;
		meter.Base.Uf               := SysPar.Gen.UfNom;
		meter.Base.If               := SysPar.Gen.IfNom;
		meter();

        //Phase Sequence
        cm0985.ClockWise            := REAL_TO_BOOL(SysPar.Gen.ClockWise);
        cm0985();

        //CM0985 - X2 and X3 - Generator
        cm0985Gen.Connection        := REAL_TO_UDINT(SysPar.Gen.Connection);
		cm0985Gen.Vprim             := SysPar.Gen.UmPrim;
		cm0985Gen.Vsec	            := SysPar.Gen.UmSec;
		cm0985Gen.Vnom		        := meter.Base.Um;
		cm0985Gen.Iprim		        := SysPar.Gen.ImPrim;
		cm0985Gen.Isec		        := REAL_TO_USINT(SysPar.Gen.ImSec);
		cm0985Gen.Inom		        := meter.Base.Im;
		cm0985Gen();
	END_IF;

	IF SysUpdate.UpdateSync THEN
		SysUpdate.UpdateSync        := FALSE;

        //Meter Base
        meter.Base.Ub               := SysPar.Sync.U1Nom;
		//CM0985 - X4 and X6 - Main
		//X4
        cm0985Main.Enable3phase     := REAL_TO_BOOL(SysPar.Sync.Enable3Phase);
        cm0985Main.Connection1      := REAL_TO_UDINT(SysPar.Sync.Connection);
		cm0985Main.V1prim			:= SysPar.Sync.U1Prim;
		cm0985Main.V1sec			:= SysPar.Sync.U1Sec;
		cm0985Main.V1nom			:= SysPar.Sync.U1Nom;
		cm0985Main();

		//CM0985 - Sync
		cm0985Sync.dFmax			:= SysPar.Sync.dFmax;
		cm0985Sync.dFmin			:= SysPar.Sync.dFmin;
		cm0985Sync.dUmax			:= SysPar.Sync.dUmax;
        cm0985Sync.UBmin            := SysPar.Sync.UBmin;
		cm0985Sync.dAngleMax		:= SysPar.Sync.dAngleMax;
		cm0985Sync.PhaseShift		:= SysPar.Sync.PhaseShift;
		cm0985Sync();

	END_IF;

	IF SysUpdate.UpdateBus THEN
		SysUpdate.UpdateBus         := FALSE;
		//CM0985 - X5 - Bus
		cm0985Bus.Vprim				:= SysPar.Exc.UexcPrim;
		cm0985Bus.Vsec				:= SysPar.Exc.UexcSec;
		cm0985Bus.Vnom				:= SysPar.Exc.UexcSec;
		cm0985Bus();
	END_IF;

	IF SysUpdate.ResetRunningHourMeter THEN
		SysUpdate.ResetRunningHourMeter	:= FALSE;
		hour_running.reset				:= TRUE;
	END_IF;

	IF SysUpdate.ResetOnlineHourMeter THEN
		SysUpdate.ResetOnlineHourMeter	:= FALSE;
		hour_online.reset				:= TRUE;
	END_IF;

	IF SysUpdate.ResetEnergy THEN
		SysUpdate.ResetEnergy			:= FALSE;
		energy_active.reset				:= TRUE;
		energy_reactive.reset			:= TRUE;
	END_IF;

    IF SysUpdate.UpdateIO THEN
		SysUpdate.UpdateIO          := FALSE;

        //AI4622
        ai4622.Channel1             := REAL_TO_UDINT(SysIOPar.AI1Type);
        ai4622.Channel2             := REAL_TO_UDINT(SysIOPar.AI2Type);
        ai4622.Channel3             := REAL_TO_UDINT(SysIOPar.AI3Type);
        ai4622.Channel4             := REAL_TO_UDINT(SysIOPar.AI4Type);
        ai4622();

        //AO4622
        ao4622.Channel1             := REAL_TO_UDINT(SysIOPar.AO1Type);
        ao4622.Channel2             := REAL_TO_UDINT(SysIOPar.AO2Type);
        ao4622.Channel3             := REAL_TO_UDINT(SysIOPar.AO3Type);
        ao4622.Channel4             := REAL_TO_UDINT(SysIOPar.AO4Type);
	    ao4622();
	END_IF;

	// Update Meters
	MdbMeter[0]	 	:= meter.In.Fm;
	MdbMeter[1]	 	:= cm0985Meter.Ug1;
	MdbMeter[2]	 	:= cm0985Meter.Ug2;
	MdbMeter[3]	 	:= cm0985Meter.Ug3;
	MdbMeter[4]	 	:= cm0985Meter.Ug12;
	MdbMeter[5]	 	:= cm0985Meter.Ug23;
	MdbMeter[6]	 	:= cm0985Meter.Ug31;
	MdbMeter[7]	 	:= cm0985Meter.Ug;
	IF cm0985Meter.Ig > 5 THEN
		MdbMeter[8]	 	:= cm0985Meter.Ig1;
		MdbMeter[9]		:= cm0985Meter.Ig2;
		MdbMeter[10] 	:= cm0985Meter.Ig3;
		MdbMeter[11] 	:= cm0985Meter.Ig;
	ELSE
		MdbMeter[8]	 	:= 0;
		MdbMeter[9]		:= 0;
		MdbMeter[10] 	:= 0;
		MdbMeter[11] 	:= 0;
	END_IF;

	MdbMeter[12] 	:= cm0985Meter.Ign;
	MdbMeter[13] 	:= cm0985Meter.Igm_dyn;
	MdbMeter[14] 	:= cm0985Meter.Pg;
	MdbMeter[15] 	:= cm0985Meter.Qg;
	MdbMeter[16] 	:= cm0985Meter.Sg;
	MdbMeter[17] 	:= meter.In.PF;
    //Exc
	MdbMeter[18]    := uf_input;
	MdbMeter[19] 	:= filter_uf.y; //meter.In.Uf;
	MdbMeter[20]    := if_input;
	MdbMeter[21] 	:= meter.In.If;
	MdbMeter[22] 	:= cm0985Meter.Fb;
	MdbMeter[23] 	:= cm0985Meter.Ub12;
	MdbMeter[24] 	:= cm0985Meter.Ub23;
	MdbMeter[25] 	:= cm0985Meter.Ub31;
    //Bus
	MdbMeter[26] 	:= cm0985Meter.Un1;
	MdbMeter[27] 	:= cm0985Meter.Un2;
	MdbMeter[28] 	:= cm0985Meter.Un3;
	MdbMeter[29] 	:= cm0985Meter.Un12;
	MdbMeter[30] 	:= cm0985Meter.Un23;
	MdbMeter[31] 	:= cm0985Meter.Un31;
	MdbMeter[32] 	:= cm0985Meter.Fs1;
	IF cm0985Meter.dAngle > 180 THEN
		MdbMeter[33]:= cm0985Meter.dAngle - 360;
	ELSE
		MdbMeter[33]:= cm0985Meter.dAngle;
	END_IF
    //Turbine
	MdbMeter[34] 	:= meter.In.Rot;
	MdbMeter[35] 	:= pos1_input;
	MdbMeter[36] 	:= pos1.PosIn;
	MdbMeter[37] 	:= pos2_input;
	MdbMeter[38] 	:= pos2.PosIn;
	MdbMeter[39] 	:= pos3_input;
	MdbMeter[40] 	:= pos3.PosIn;
    //
	MdbMeter[41] 	:= ExcTemp;												//Excitation Temperature
	MdbMeter[42]	:= hour_running.horas;
	MdbMeter[43]	:= hour_running.minutos;
	MdbMeter[44]	:= hour_online.horas;
	MdbMeter[45]	:= hour_online.minutos;
	MdbMeter[46]	:= LREAL_TO_REAL(energy_active.posEnergy);
	MdbMeter[47]	:= LREAL_TO_REAL(energy_active.negEnergy);
	MdbMeter[48]	:= LREAL_TO_REAL(energy_reactive.posEnergy);
	MdbMeter[49]	:= LREAL_TO_REAL(energy_reactive.negEnergy);

END_PROGRAM
```

- Cyclic.st.bak (not shown)

#### Init.st
```iecst
PROGRAM _INIT
    TagManager(enable:=TRUE);
    //Register Parameters
    PgsTagStartNode     (TagManager.ident, ADR('system'));
    //Sync
    PgsTagStartNode     (TagManager.ident, ADR('sync'));
    PgsTagRegisterREAL  (TagManager.ident, TRUE, ADR('U1Prim'),         SysPar.Sync.U1Prim);
    PgsTagRegisterREAL  (TagManager.ident, TRUE, ADR('U1Sec'),          SysPar.Sync.U1Sec);
    PgsTagRegisterREAL  (TagManager.ident, TRUE, ADR('Enable3Phase'),   SysPar.Sync.Enable3Phase);
    PgsTagRegisterREAL  (TagManager.ident, TRUE, ADR('Connection'),     SysPar.Sync.Connection);
    PgsTagRegisterREAL  (TagManager.ident, TRUE, ADR('U1Nom'),          SysPar.Sync.U1Nom);
    PgsTagRegisterREAL  (TagManager.ident, TRUE, ADR('UBmin'),          SysPar.Sync.UBmin);
    PgsTagRegisterREAL  (TagManager.ident, TRUE, ADR('dFmax'),          SysPar.Sync.dFmax);
    PgsTagRegisterREAL  (TagManager.ident, TRUE, ADR('dFmin'),          SysPar.Sync.dFmin);
    PgsTagRegisterREAL  (TagManager.ident, TRUE, ADR('dUmax'),          SysPar.Sync.dUmax);
    PgsTagRegisterREAL  (TagManager.ident, TRUE, ADR('dAngleMax'),      SysPar.Sync.dAngleMax);
    PgsTagRegisterREAL  (TagManager.ident, TRUE, ADR('PhaseShift'),     SysPar.Sync.PhaseShift);
    PgsTagEndNode       (TagManager.ident);//sync
    //Bus
    PgsTagStartNode     (TagManager.ident, ADR('exc'));
    PgsTagRegisterREAL  (TagManager.ident, TRUE, ADR('UexcPrim'),     SysPar.Exc.UexcPrim);
    PgsTagRegisterREAL  (TagManager.ident, TRUE, ADR('UexcSec'),      SysPar.Exc.UexcSec);
    PgsTagRegisterREAL  (TagManager.ident, TRUE, ADR('UexcNom'),      SysPar.Exc.UexcNom);
    PgsTagEndNode       (TagManager.ident);//bus
    //Gen
    PgsTagStartNode     (TagManager.ident, ADR('gen'));
    PgsTagRegisterREAL  (TagManager.ident, TRUE, ADR('UmPrim'),     SysPar.Gen.UmPrim);
    PgsTagRegisterREAL  (TagManager.ident, TRUE, ADR('UmSec'),      SysPar.Gen.UmSec);
    PgsTagRegisterREAL  (TagManager.ident, TRUE, ADR('ImPrim'),     SysPar.Gen.ImPrim);
    PgsTagRegisterREAL  (TagManager.ident, TRUE, ADR('ImSec'),      SysPar.Gen.ImSec);
    PgsTagRegisterREAL  (TagManager.ident, TRUE, ADR('UmNom'),      SysPar.Gen.UmNom);
    PgsTagRegisterREAL  (TagManager.ident, TRUE, ADR('SmNom'),      SysPar.Gen.SmNom);
    PgsTagRegisterREAL  (TagManager.ident, TRUE, ADR('FmNom'),      SysPar.Gen.FmNom);
    PgsTagRegisterREAL  (TagManager.ident, TRUE, ADR('UfMin'),      SysPar.Gen.UfMin);
    PgsTagRegisterREAL  (TagManager.ident, TRUE, ADR('UfMax'),      SysPar.Gen.UfMax);
    PgsTagRegisterREAL  (TagManager.ident, TRUE, ADR('UfNom'),      SysPar.Gen.UfNom);
    PgsTagRegisterREAL  (TagManager.ident, TRUE, ADR('IfMin'),      SysPar.Gen.IfMin);
    PgsTagRegisterREAL  (TagManager.ident, TRUE, ADR('IfMax'),      SysPar.Gen.IfMax);
    PgsTagRegisterREAL  (TagManager.ident, TRUE, ADR('IfNom'),      SysPar.Gen.IfNom);
    PgsTagRegisterREAL  (TagManager.ident, TRUE, ADR('RpmNom'),     SysPar.Gen.RpmNom);
    PgsTagRegisterREAL  (TagManager.ident, TRUE, ADR('PPR1'),       SysPar.Gen.PPR1);
    PgsTagRegisterREAL  (TagManager.ident, TRUE, ADR('Pos1_0p'),    SysPar.Gen.Pos1_0p);
    PgsTagRegisterREAL  (TagManager.ident, TRUE, ADR('Pos1_100p'),  SysPar.Gen.Pos1_100p);
    PgsTagRegisterREAL  (TagManager.ident, TRUE, ADR('Pos2_0p'),    SysPar.Gen.Pos2_0p);
    PgsTagRegisterREAL  (TagManager.ident, TRUE, ADR('Pos2_100p'),  SysPar.Gen.Pos2_100p);
    PgsTagRegisterREAL  (TagManager.ident, TRUE, ADR('Pos3_0p'),    SysPar.Gen.Pos3_0p);
    PgsTagRegisterREAL  (TagManager.ident, TRUE, ADR('Pos3_100p'),  SysPar.Gen.Pos3_100p);
    PgsTagRegisterREAL  (TagManager.ident, TRUE, ADR('ClockWise'),  SysPar.Gen.ClockWise);
    PgsTagRegisterREAL  (TagManager.ident, TRUE, ADR('Connection'), SysPar.Gen.Connection);
    PgsTagRegisterREAL  (TagManager.ident, TRUE, ADR('dRpm1Max'),   SysPar.Gen.dRpm1Max);
    PgsTagRegisterREAL  (TagManager.ident, TRUE, ADR('PPR2'),       SysPar.Gen.PPR2);
    PgsTagRegisterREAL  (TagManager.ident, TRUE, ADR('dRpm2Max'),   SysPar.Gen.dRpm2Max);
    PgsTagEndNode       (TagManager.ident);//gen
    //IO
    PgsTagStartNode     (TagManager.ident, ADR('io'));
    PgsTagRegisterREAL  (TagManager.ident, TRUE, ADR('AI1Type'),    SysIOPar.AI1Type);
    PgsTagRegisterREAL  (TagManager.ident, TRUE, ADR('AI2Type'),    SysIOPar.AI2Type);
    PgsTagRegisterREAL  (TagManager.ident, TRUE, ADR('AI3Type'),    SysIOPar.AI3Type);
    PgsTagRegisterREAL  (TagManager.ident, TRUE, ADR('AI4Type'),    SysIOPar.AI4Type);
    PgsTagRegisterREAL  (TagManager.ident, TRUE, ADR('AO1Type'),    SysIOPar.AO1Type);
    PgsTagRegisterREAL  (TagManager.ident, TRUE, ADR('AO2Type'),    SysIOPar.AO2Type);
    PgsTagRegisterREAL  (TagManager.ident, TRUE, ADR('AO3Type'),    SysIOPar.AO3Type);
    PgsTagRegisterREAL  (TagManager.ident, TRUE, ADR('AO4Type'),    SysIOPar.AO4Type);
    PgsTagRegisterREAL  (TagManager.ident, TRUE, ADR('AO1min'),     SysIOPar.AO1min);
    PgsTagRegisterREAL  (TagManager.ident, TRUE, ADR('AO1max'),     SysIOPar.AO1max);
    PgsTagRegisterREAL  (TagManager.ident, TRUE, ADR('AO2min'),     SysIOPar.AO2min);
    PgsTagRegisterREAL  (TagManager.ident, TRUE, ADR('AO2max'),     SysIOPar.AO2max);
    PgsTagRegisterREAL  (TagManager.ident, TRUE, ADR('AO3min'),     SysIOPar.AO3min);
    PgsTagRegisterREAL  (TagManager.ident, TRUE, ADR('AO3max'),     SysIOPar.AO3max);
    PgsTagRegisterREAL  (TagManager.ident, TRUE, ADR('AO4min'),     SysIOPar.AO4min);
    PgsTagRegisterREAL  (TagManager.ident, TRUE, ADR('AO4max'),     SysIOPar.AO4max);
    PgsTagEndNode       (TagManager.ident);//io
    PgsTagEndNode       (TagManager.ident);//system

    SysUpdate.UpdateAll := TRUE;

	//Horimetro
    PgsTagStartNode     (TagManager.ident, ADR('Horimetro'));
    PgsTagRegisterREAL  (TagManager.ident, TRUE, ADR('running_total'),	hour_running.set_total);
    PgsTagRegisterREAL  (TagManager.ident, TRUE, ADR('online_total'),	hour_online.set_total);
	PgsTagEndNode       (TagManager.ident);//Horimetro

	//Energia
    PgsTagStartNode     (TagManager.ident, ADR('Energia'));
    PgsTagRegisterREAL  (TagManager.ident, TRUE, ADR('ativa_pos'),				energy_active.set_posEnergy);
    PgsTagRegisterREAL  (TagManager.ident, TRUE, ADR('ativa_neg'),				energy_active.set_negEnergy);
    PgsTagRegisterREAL  (TagManager.ident, TRUE, ADR('reativa_pos'),			energy_reactive.set_posEnergy);
    PgsTagRegisterREAL  (TagManager.ident, TRUE, ADR('reativa_neg'),			energy_reactive.set_negEnergy);
	PgsTagEndNode       (TagManager.ident);//Energia

END_PROGRAM
```

- Init.st.bak (not shown)

- Variables.var.bak (not shown)

### Share.typ
```iecst
TYPE
	PgsA65 : 	STRUCT
		di : PgsA65DI;
		do : PgsA65DO;
		ai : PgsA65AI;
		ao : PgsA65AO;
	END_STRUCT;
	PgsA65DI : 	STRUCT
		remote : BOOL;
		reset : BOOL;
		gov_enable : BOOL;
		gov_ctrl_pwr_enable : BOOL;
		gov_trip : BOOL;
		gov_unload : BOOL;
		gov_up : BOOL;
		gov_down : BOOL;
		avr_enable : BOOL;
		avr_ctrl_qm_enable : BOOL;
		avr_ctrl_pf_enable : BOOL;
		avr_trip : BOOL;
		avr_unload : BOOL;
		avr_ref_up : BOOL;
		avr_ref_down : BOOL;
		sync_enable : BOOL;
		dead_bus_enable : BOOL;
		enable_pos1 : BOOL;
		enable_pos2 : BOOL;
		enable_pos3 : BOOL;
	END_STRUCT;
	PgsA65DO : 	STRUCT
		gov_on : BOOL;
		gov_unload : BOOL;
		gov_over_rotation : BOOL;
		rotation_zero : BOOL;
		rotation_nominal : BOOL;
		rotation_brake : BOOL;
		power_zero : BOOL;
		rpm_fault : BOOL;
		avr_on : BOOL;
		online : BOOL;
		avr_force_crowbar : BOOL;
		avr_limiter_on : BOOL;
		field_flash_on : BOOL;
		voltage_nominal : BOOL;
		sync_enabled : BOOL;
		dead_bus_enabled : BOOL;
		watchdog : BOOL;
	END_STRUCT;
	PgsA65AI : 	STRUCT
		if : INT;
		uf : INT;
		pos1 : INT;
		pos2 : INT;
		pos3 : INT;
	END_STRUCT;
	PgsA65AO : 	STRUCT
		pwr : INT;
		pos1 : INT;
		pos2 : INT;
		pos3 : INT;
	END_STRUCT;
END_TYPE
```

### Share.var
```iecst
(*I/O*)
VAR
	A65 : PgsA65;
END_VAR
(*Controls*)
VAR
	avr : PgsAVR := (Parameter:=(CtrlManual:=(CmIf:=(Enable:=FALSE,dRefOn:=0.1,dRefOff:=0.1,PID:=(Kp:=0.004,Ti:=0.05,Td:=0.0,Tf:=1.0,Kwd:=1.2)),CmUf:=(Enable:=FALSE,dRefOn:=0.1,dRefOff:=0.1,PID:=(Kp:=0.002,Ti:=0.05,Td:=0.0,Tf:=1.0,Kwd:=1.2)),CmIm:=(Enable:=FALSE),Ctrl:=PGS_AVR_CM_OFF,EnableOL:=FALSE),CtrlAuto:=(SoftStart:=(RefUm:=1.0,dRefOn:=0.05,dRefOff:=0.0,Offset:=0,RefUm0:=0.3948,FFTmin:=0,FFTmax:=5.0),CaUm0:=(Enable:=FALSE,Ref:=1.0,RefMax:=1.2,RefMin:=0.8,dRefOn:=0.07,dRefOff:=0.07,Kdp:=0.0,PID:=(Kp:=0.003,Ti:=0.1,Td:=0.05,Tf:=1.0,Kwd:=1.2)),CaUm1:=(Enable:=FALSE),CaQm:=(Enable:=FALSE,Ref:=-0.08,RefMax:=0.5,RefMin:=-0.5,dRefOn:=0.01,dRefOff:=0.01,PID:=(Kp:=0.0006,Ti:=1.0,Td:=0.0,Tf:=1.0,Kwd:=1.2),L2max:=1.2,L2min:=0.8,Kdp:=0.1,PIDU:=(Kp:=0.002,Ti:=0.1,Td:=0.05,Tf:=1.0,Kwd:=1.2)),CaPf:=(Enable:=FALSE,Ref:=-0.1,RefMax:=0.3,RefMin:=-0.3,dRefOn:=0.05,dRefOff:=0.05,PID:=(Kp:=0.0006,Ti:=0.8,Td:=0.0,Tf:=1.0,Kwd:=1.2),L2max:=1.2,L2min:=0.8,Kdp:=0.1,PIDU:=(Kp:=0.002,Ti:=0.09,Td:=0.05,Tf:=1.0,Kwd:=1.2))),Limiter:=(Luh:=(Enable:=FALSE,Un:=1.0,Fn:=0.98,Kuh:=1.0,PID:=(Kp:=0.003,Ti:=0.1,Td:=0.05,Tf:=1.0,Kwd:=1.2)),Lifh:=(Enable:=FALSE,SetPoint:=1.1312,Curve:=PGS_AVR_CV_00,Time:=10.0,PID:=(Kp:=0.004,Ti:=0.05,Td:=0.0,Tf:=1.0,Kwd:=1.2)),Lifl:=(Enable:=FALSE,SetPoint:=0.2262,PID:=(Kp:=0.004,Ti:=0.05,Td:=0.0,Tf:=1.0,Kwd:=1.2)),Lifhh:=(Enable:=FALSE,SetPoint:=1.3574,PID:=(Kp:=0.004,Ti:=0.05,Td:=0.0,Tf:=1.0,Kwd:=1.2)),Limh:=(Enable:=FALSE),Lpq:=(Enable:=FALSE))),CtrlOnline:=PGS_AVR_CA_PF);
	gov : PgsGOV := (Parameter:=(CtrlManual:=(CmPos:=(Enable:=FALSE,dRefOn:=0.1,dRefOff:=0.1,RefMax:=1.0,RefMin:=0.0)),CtrlAuto:=(SoftStart:=(Pos0:=0.25,dPos:=0.1,Rpm0:=0.0,Rpm1:=0.2,Rpm2:=0.8,RpmBrake:=0.0,dRpmOn:=0.05,dRpmOff:=0.05,TRpm1:=120,TRpm2:=300),CaRpm0:=(Enable:=FALSE,Ref:=1.0,RefMax:=1.2,RefMin:=0.0,dRefOn:=0.05,dRefOff:=0.05,Kdp:=0.0,PosMax:=0.95,PID:=(Kp:=0.003,Ti:=0.15,Td:=0.0,Tf:=1.0,Kwd:=1.0)),CaRpm1:=(Enable:=FALSE,Ref:=1.025,RefMax:=1.1,RefMin:=0.9,dRefOn:=0.01,dRefOff:=0.01,Kdp:=0.1,PosMax:=0.95,PID:=(Kp:=0.003,Ti:=0.15,Td:=0.0,Tf:=1.0,Kwd:=1.0)),CaHz0:=(Enable:=FALSE,UmOn:=0.5,Ref:=1.0,RefMax:=1.2,RefMin:=0.9,dRefOn:=0.01,dRefOff:=0.1,Kdp:=0.0,PosMax:=0.95,PID:=(Kp:=0.002,Ti:=0.2,Td:=0.5,Tf:=1.0,Kwd:=1.0)),CaHz1:=(Enable:=FALSE,UmOn:=0.5,Ref:=1.025,RefMax:=1.2,RefMin:=0.9,dRefOn:=0.01,dRefOff:=0.01,Kdp:=0.1,PosMax:=0.95,PID:=(Kp:=0.003,Ti:=0.15,Td:=0.0,Tf:=1.0,Kwd:=1.0)),CaPwr:=(Enable:=FALSE,UmOn:=0.5,Ref:=0.02,RefMax:=1.05,RefMin:=0.0,dRefOn:=0.01,dRefOff:=0.01,PID:=(Kp:=0.001,Ti:=0.8,Td:=0.0,Tf:=1.0,Kwd:=1.0),L2max:=1.1,L2min:=0.9,Kdp:=0.1,PosMax:=0.8,PIDHz:=(Kp:=0.002,Ti:=0.2,Td:=0.5,Tf:=1.0,Kwd:=1.0)))),CtrlOnline:=PGS_GOV_CA_PWR);
	pos1 : PgsPOS := (Parameter:=(Enable:=FALSE,Base:=100,RampUp:=(dSp0:=0.1,SetPoint:=0.2,dSp1:=0.3),RampDown:=(dSp0:=0.05,SetPoint:=0.15,dSp1:=0.2),HCC:=(Kup:=1.0,Kdown:=1.0,dbHigh:=0.55,dbLow:=0.45),PID:=(Kp:=0.05,Ti:=5.0,Td:=0.0,Tf:=1.0,Kwd:=1.0,Update:=TRUE)));
	pos2 : PgsPOS := (Parameter:=(Enable:=FALSE,Base:=100,RampUp:=(dSp0:=0.1,SetPoint:=0.2,dSp1:=0.3),RampDown:=(dSp0:=0.05,SetPoint:=0.15,dSp1:=0.2),HCC:=(Kup:=1.0,Kdown:=1.0,dbHigh:=0.55,dbLow:=0.45),PID:=(Kp:=0.05,Ti:=5.0,Td:=0.0,Tf:=1.0,Kwd:=1.0,Update:=TRUE)));
	pos3 : PgsPOS := (Parameter:=(Enable:=FALSE,Base:=100,RampUp:=(dSp0:=0.1,SetPoint:=0.2,dSp1:=0.3),RampDown:=(dSp0:=0.05,SetPoint:=0.15,dSp1:=0.2),HCC:=(Kup:=1.0,Kdown:=1.0,dbHigh:=0.55,dbLow:=0.45),PID:=(Kp:=0.05,Ti:=5.0,Td:=0.0,Tf:=1.0,Kwd:=1.0,Update:=TRUE)));
	curve1 : PgsCurve := (Curve:=(in:=[0.0,0.2,0.3,0.4,0.5,0.6,0.7,0.8,0.9,1.0],out:=[0.0,0.2,0.3,0.4,0.5,0.6,0.7,0.8,0.9,1.0]));
	curve2 : PgsCurve := (Curve:=(in:=[0.0,0.2,0.3,0.4,0.5,0.6,0.7,0.8,0.9,1.0],out:=[0.0,0.2,0.3,0.4,0.5,0.6,0.7,0.8,0.9,1.0]));
	curve3 : PgsCurve := (Curve:=(in:=[0.0,0.2,0.3,0.4,0.5,0.6,0.7,0.8,0.9,1.0],out:=[0.0,0.2,0.3,0.4,0.5,0.6,0.7,0.8,0.9,1.0]));
END_VAR
(*Protection*)
VAR
	phaseFault : PgsProtPhaseFault;
END_VAR
(*Meter*)
VAR
	meter : PgsMeter := (Base:=(Sm:=1000,Um:=380,Fm:=60,Rot:=2000,Uf:=80,If:=10));
	filter_uf : LCRMovAvgFlt;
	pos1_input : REAL;
	pos2_input : REAL;
	pos3_input : REAL;
	uf_input : REAL;
	if_input : REAL;
END_VAR
(*Hour Meter*)
VAR
	hour_running : PgsHorimetro;
	hour_online : PgsHorimetro;
END_VAR
(*Energy Meter*)
VAR
	energy_active : PgsEnergia;
	energy_reactive : PgsEnergia;
END_VAR
```

- Share.typ.bak (not shown)

### Program Logical/Kontrol/Control/Control

#### Variables.var
```iecst
(*PWR*)
VAR
	pwr_tp : TP;
	pwr_ton : TON;
	pwr_mem : BOOL;
	filter_pwr : PgsFiltro := (CTE:=100);
END_VAR
(*RPM*)
VAR
	rpm1 : PgsRPM;
	rpm2 : PgsRPM;
	filter_rpm1 : PgsFiltro;
	filter_rpm2 : PgsFiltro;
END_VAR
(*Analog Inputs*)
VAR
	scale_if : LCRScal;
	scale_uf : LCRScal;
	scale_pos1 : LCRScal;
	scale_pos2 : LCRScal;
	scale_pos3 : LCRScal;
	filter_pos1 : PgsFiltro := (CTE:=20);
END_VAR
(*Analog Outputs*)
VAR
	scale_avr_o1 : LCRScal;
	scale_gov_o1 : LCRScal;
	scale_gov_o2 : LCRScal;
	scale_gov_o3 : LCRScal;
END_VAR
```
